	UF : 1, UT : 1,		CONFIG : 'N U T, 0, 0, 1',
	X =  25.000  mm,	Y =  64.000  mm,	Z =   15.000 mm,
	W =180.000 deg,	P =   0.000 deg,	R =    90.000 deg
};
P[3598]{
   GP1:
	UF : 1, UT : 1,		CONFIG : 'N U T, 0, 0, 1',
	X =  31.000  mm,	Y =  64.000  mm,	Z =   15.000 mm,
	W =180.000 deg,	P =   0.000 deg,	R =    90.000 deg
};
P[3599]{
   GP1:
	UF : 1, UT : 1,		CONFIG : 'N U T, 0, 0, 1',
	X =  31.000  mm,	Y =  64.000  mm,	Z =   0.600 mm,
	W =180.000 deg,	P =   0.000 deg,	R =    90.000 deg
};
P[3600]{
   GP1:
	UF : 1, UT : 1,		CONFIG : 'N U T, 0, 0, 1',
	X =  31.000  mm,	Y =  64.000  mm,	Z =   15.000 mm,
	W =180.000 deg,	P =   0.000 deg,	R =    90.000 deg
};
P[3601]{
   GP1:
	UF : 1, UT : 1,		CONFIG : 'N U T, 0, 0, 1',
	X =  34.000  mm,	Y =  64.000  mm,	Z =   15.000 mm,
	W =180.000 deg,	P =   0.000 deg,	R =    90.000 deg
};
P[3602]{
   GP1:
	UF : 1, UT : 1,		CONFIG : 'N U T, 0, 0, 1',
	X =  34.000  mm,	Y =  64.000  mm,	Z =   0.600 mm,
	W =180.000 deg,	P =   0.000 deg,	R =    90.000 deg
};
P[3603]{
   GP1:
	UF : 1, UT : 1,		CONFIG : 'N U T, 0, 0, 1',
	X =  34.000  mm,	Y =  64.000  mm,	Z =   15.000 mm,
	W =180.000 deg,	P =   0.000 deg,	R =    90.000 deg
};
P[3604]{
   GP1:
	UF : 1, UT : 1,		CONFIG : 'N U T, 0, 0, 1',
	X =  37.000  mm,	Y =  64.000  mm,	Z =   15.000 mm,
	W =180.000 deg,	P =   0.000 deg,	R =    90.000 deg
};
P[3605]{
   GP1:
	UF : 1, UT : 1,		CONFIG : 'N U T, 0, 0, 1',
	X =  37.000  mm,	Y =  64.000  mm,	Z =   0.600 mm,
	W =180.000 deg,	P =   0.000 deg,	R =    90.000 deg
};
P[3606]{
   GP1:
	UF : 1, UT : 1,		CONFIG : 'N U T, 0, 0, 1',
	X =  37.000  mm,	Y =  64.000  mm,	Z =   15.000 mm,
	W =180.000 deg,	P =   0.000 deg,	R =    90.000 deg
};
P[3607]{
   GP1:
	UF : 1, UT : 1,		CONFIG : 'N U T, 0, 0, 1',
	X =  40.000  mm,	Y =  64.000  mm,	Z =   15.000 mm,
	W =180.000 deg,	P =   0.000 deg,	R =    90.000 deg
};
P[3608]{
   GP1:
	UF : 1, UT : 1,		CONFIG : 'N U T, 0, 0, 1',
	X =  40.000  mm,	Y =  64.000  mm,	Z =   0.600 mm,
	W =180.000 deg,	P =   0.000 deg,	R =    90.000 deg
};
P[3609]{
   GP1:
	UF : 1, UT : 1,		CONFIG : 'N U T, 0, 0, 1',
	X =  40.000  mm,	Y =  64.000  mm,	Z =   15.000 mm,
	W =180.000 deg,	P =   0.000 deg,	R =    90.000 deg
};
P[3610]{
   GP1:
	UF : 1, UT : 1,		CONFIG : 'N U T, 0, 0, 1',
	X =  43.000  mm,	Y =  64.000  mm,	Z =   15.000 mm,
	W =180.000 deg,	P =   0.000 deg,	R =    90.000 deg
};
P[3611]{
   GP1:
	UF : 1, UT : 1,		CONFIG : 'N U T, 0, 0, 1',
	X =  43.000  mm,	Y =  64.000  mm,	Z =   0.600 mm,
	W =180.000 deg,	P =   0.000 deg,	R =    90.000 deg
};
P[3612]{
   GP1:
	UF : 1, UT : 1,		CONFIG : 'N U T, 0, 0, 1',
	X =  43.000  mm,	Y =  64.000  mm,	Z =   15.000 mm,
	W =180.000 deg,	P =   0.000 deg,	R =    90.000 deg
};
P[3613]{
   GP1:
	UF : 1, UT : 1,		CONFIG : 'N U T, 0, 0, 1',
	X =  46.000  mm,	Y =  64.000  mm,	Z =   15.000 mm,
	W =180.000 deg,	P =   0.000 deg,	R =    90.000 deg
};
P[3614]{
   GP1:
	UF : 1, UT : 1,		CONFIG : 'N U T, 0, 0, 1',
	X =  46.000  mm,	Y =  64.000  mm,	Z =   0.600 mm,
	W =180.000 deg,	P =   0.000 deg,	R =    90.000 deg
};
P[3615]{
   GP1:
	UF : 1, UT : 1,		CONFIG : 'N U T, 0, 0, 1',
	X =  46.000  mm,	Y =  64.000  mm,	Z =   15.000 mm,
	W =180.000 deg,	P =   0.000 deg,	R =    90.000 deg
};
P[3616]{
   GP1:
	UF : 1, UT : 1,		CONFIG : 'N U T, 0, 0, 1',
	X =  49.000  mm,	Y =  64.000  mm,	Z =   15.000 mm,
	W =180.000 deg,	P =   0.000 deg,	R =    90.000 deg
};
P[3617]{
   GP1:
	UF : 1, UT : 1,		CONFIG : 'N U T, 0, 0, 1',
	X =  49.000  mm,	Y =  64.000  mm,	Z =   0.600 mm,
	W =180.000 deg,	P =   0.000 deg,	R =    90.000 deg
};
P[3618]{
   GP1:
	UF : 1, UT : 1,		CONFIG : 'N U T, 0, 0, 1',
	X =  49.000  mm,	Y =  64.000  mm,	Z =   15.000 mm,
	W =180.000 deg,	P =   0.000 deg,	R =    90.000 deg
};
P[3619]{
   GP1:
	UF : 1, UT : 1,		CONFIG : 'N U T, 0, 0, 1',
	X =  52.000  mm,	Y =  64.000  mm,	Z =   15.000 mm,
	W =180.000 deg,	P =   0.000 deg,	R =    90.000 deg
};
P[3620]{
   GP1:
	UF : 1, UT : 1,		CONFIG : 'N U T, 0, 0, 1',
	X =  52.000  mm,	Y =  64.000  mm,	Z =   0.600 mm,
	W =180.000 deg,	P =   0.000 deg,	R =    90.000 deg
};
P[3621]{
   GP1:
	UF : 1, UT : 1,		CONFIG : 'N U T, 0, 0, 1',
	X =  52.000  mm,	Y =  64.000  mm,	Z =   15.000 mm,
	W =180.000 deg,	P =   0.000 deg,	R =    90.000 deg
};
P[3622]{
   GP1:
	UF : 1, UT : 1,		CONFIG : 'N U T, 0, 0, 1',
	X =  55.000  mm,	Y =  64.000  mm,	Z =   15.000 mm,
	W =180.000 deg,	P =   0.000 deg,	R =    90.000 deg
};
P[3623]{
   GP1:
	UF : 1, UT : 1,		CONFIG : 'N U T, 0, 0, 1',
	X =  55.000  mm,	Y =  64.000  mm,	Z =   0.600 mm,
	W =180.000 deg,	P =   0.000 deg,	R =    90.000 deg
};
P[3624]{
   GP1:
	UF : 1, UT : 1,		CONFIG : 'N U T, 0, 0, 1',
	X =  55.000  mm,	Y =  64.000  mm,	Z =   15.000 mm,
	W =180.000 deg,	P =   0.000 deg,	R =    90.000 deg
};
P[3628]{
   GP1:
	UF : 1, UT : 1,		CONFIG : 'N U T, 0, 0, 1',
	X =  61.000  mm,	Y =  64.000  mm,	Z =   15.000 mm,
	W =180.000 deg,	P =   0.000 deg,	R =    90.000 deg
};
P[3629]{
   GP1:
	UF : 1, UT : 1,		CONFIG : 'N U T, 0, 0, 1',
	X =  61.000  mm,	Y =  64.000  mm,	Z =   0.600 mm,
	W =180.000 deg,	P =   0.000 deg,	R =    90.000 deg
};
P[3630]{
   GP1:
	UF : 1, UT : 1,		CONFIG : 'N U T, 0, 0, 1',
	X =  61.000  mm,	Y =  64.000  mm,	Z =   15.000 mm,
	W =180.000 deg,	P =   0.000 deg,	R =    90.000 deg
};
P[3649]{
   GP1:
	UF : 1, UT : 1,		CONFIG : 'N U T, 0, 0, 1',
	X =  82.000  mm,	Y =  64.000  mm,	Z =   15.000 mm,
	W =180.000 deg,	P =   0.000 deg,	R =    90.000 deg
};
P[3650]{
   GP1:
	UF : 1, UT : 1,		CONFIG : 'N U T, 0, 0, 1',
	X =  82.000  mm,	Y =  64.000  mm,	Z =   0.600 mm,
	W =180.000 deg,	P =   0.000 deg,	R =    90.000 deg
};
P[3651]{
   GP1:
	UF : 1, UT : 1,		CONFIG : 'N U T, 0, 0, 1',
	X =  82.000  mm,	Y =  64.000  mm,	Z =   15.000 mm,
	W =180.000 deg,	P =   0.000 deg,	R =    90.000 deg
};
P[3652]{
   GP1:
	UF : 1, UT : 1,		CONFIG : 'N U T, 0, 0, 1',
	X =  85.000  mm,	Y =  64.000  mm,	Z =   15.000 mm,
	W =180.000 deg,	P =   0.000 deg,	R =    90.000 deg
};
P[3653]{
   GP1:
	UF : 1, UT : 1,		CONFIG : 'N U T, 0, 0, 1',
	X =  85.000  mm,	Y =  64.000  mm,	Z =   0.600 mm,
	W =180.000 deg,	P =   0.000 deg,	R =    90.000 deg
};
P[3654]{
   GP1:
	UF : 1, UT : 1,		CONFIG : 'N U T, 0, 0, 1',
	X =  85.000  mm,	Y =  64.000  mm,	Z =   15.000 mm,
	W =180.000 deg,	P =   0.000 deg,	R =    90.000 deg
};
P[3655]{
   GP1:
	UF : 1, UT : 1,		CONFIG : 'N U T, 0, 0, 1',
	X =  88.000  mm,	Y =  64.000  mm,	Z =   15.000 mm,
	W =180.000 deg,	P =   0.000 deg,	R =    90.000 deg
};
P[3656]{
   GP1:
	UF : 1, UT : 1,		CONFIG : 'N U T, 0, 0, 1',
	X =  88.000  mm,	Y =  64.000  mm,	Z =   0.600 mm,
	W =180.000 deg,	P =   0.000 deg,	R =    90.000 deg
};
P[3657]{
   GP1:
	UF : 1, UT : 1,		CONFIG : 'N U T, 0, 0, 1',
	X =  88.000  mm,	Y =  64.000  mm,	Z =   15.000 mm,
	W =180.000 deg,	P =   0.000 deg,	R =    90.000 deg
};
P[3658]{
   GP1:
	UF : 1, UT : 1,		CONFIG : 'N U T, 0, 0, 1',
	X =  91.000  mm,	Y =  64.000  mm,	Z =   15.000 mm,
	W =180.000 deg,	P =   0.000 deg,	R =    90.000 deg
};
P[3659]{
   GP1:
	UF : 1, UT : 1,		CONFIG : 'N U T, 0, 0, 1',
	X =  91.000  mm,	Y =  64.000  mm,	Z =   0.600 mm,
	W =180.000 deg,	P =   0.000 deg,	R =    90.000 deg
};
P[3660]{
   GP1:
	UF : 1, UT : 1,		CONFIG : 'N U T, 0, 0, 1',
	X =  91.000  mm,	Y =  64.000  mm,	Z =   15.000 mm,
	W =180.000 deg,	P =   0.000 deg,	R =    90.000 deg
};
P[3661]{
   GP1:
	UF : 1, UT : 1,		CONFIG : 'N U T, 0, 0, 1',
	X =  94.000  mm,	Y =  64.000  mm,	Z =   15.000 mm,
	W =180.000 deg,	P =   0.000 deg,	R =    90.000 deg
};
P[3662]{
   GP1:
	UF : 1, UT : 1,		CONFIG : 'N U T, 0, 0, 1',
	X =  94.000  mm,	Y =  64.000  mm,	Z =   0.600 mm,
	W =180.000 deg,	P =   0.000 deg,	R =    90.000 deg
};
P[3663]{
   GP1:
	UF : 1, UT : 1,		CONFIG : 'N U T, 0, 0, 1',
	X =  94.000  mm,	Y =  64.000  mm,	Z =   15.000 mm,
	W =180.000 deg,	P =   0.000 deg,	R =    90.000 deg
};
P[3664]{
   GP1:
	UF : 1, UT : 1,		CONFIG : 'N U T, 0, 0, 1',
	X =  97.000  mm,	Y =  64.000  mm,	Z =   15.000 mm,
	W =180.000 deg,	P =   0.000 deg,	R =    90.000 deg
};
P[3665]{
   GP1:
	UF : 1, UT : 1,		CONFIG : 'N U T, 0, 0, 1',
	X =  97.000  mm,	Y =  64.000  mm,	Z =   0.600 mm,
	W =180.000 deg,	P =   0.000 deg,	R =    90.000 deg
};
P[3666]{
   GP1:
	UF : 1, UT : 1,		CONFIG : 'N U T, 0, 0, 1',
	X =  97.000  mm,	Y =  64.000  mm,	Z =   15.000 mm,
	W =180.000 deg,	P =   0.000 deg,	R =    90.000 deg
};
P[3667]{
   GP1:
	UF : 1, UT : 1,		CONFIG : 'N U T, 0, 0, 1',
	X =  100.000  mm,	Y =  64.000  mm,	Z =   15.000 mm,
	W =180.000 deg,	P =   0.000 deg,	R =    90.000 deg
};
P[3668]{
   GP1:
	UF : 1, UT : 1,		CONFIG : 'N U T, 0, 0, 1',
	X =  100.000  mm,	Y =  64.000  mm,	Z =   0.600 mm,
	W =180.000 deg,	P =   0.000 deg,	R =    90.000 deg
};
P[3669]{
   GP1:
	UF : 1, UT : 1,		CONFIG : 'N U T, 0, 0, 1',
	X =  100.000  mm,	Y =  64.000  mm,	Z =   15.000 mm,
	W =180.000 deg,	P =   0.000 deg,	R =    90.000 deg
};
P[3670]{
   GP1:
	UF : 1, UT : 1,		CONFIG : 'N U T, 0, 0, 1',
	X =  103.000  mm,	Y =  64.000  mm,	Z =   15.000 mm,
	W =180.000 deg,	P =   0.000 deg,	R =    90.000 deg
};
P[3671]{
   GP1:
	UF : 1, UT : 1,		CONFIG : 'N U T, 0, 0, 1',
	X =  103.000  mm,	Y =  64.000  mm,	Z =   0.600 mm,
	W =180.000 deg,	P =   0.000 deg,	R =    90.000 deg
};
P[3672]{
   GP1:
	UF : 1, UT : 1,		CONFIG : 'N U T, 0, 0, 1',
	X =  103.000  mm,	Y =  64.000  mm,	Z =   15.000 mm,
	W =180.000 deg,	P =   0.000 deg,	R =    90.000 deg
};
P[3673]{
   GP1:
	UF : 1, UT : 1,		CONFIG : 'N U T, 0, 0, 1',
	X =  106.000  mm,	Y =  64.000  mm,	Z =   15.000 mm,
	W =180.000 deg,	P =   0.000 deg,	R =    90.000 deg
};
P[3674]{
   GP1:
	UF : 1, UT : 1,		CONFIG : 'N U T, 0, 0, 1',
	X =  106.000  mm,	Y =  64.000  mm,	Z =   0.600 mm,
	W =180.000 deg,	P =   0.000 deg,	R =    90.000 deg
};
P[3675]{
   GP1:
	UF : 1, UT : 1,		CONFIG : 'N U T, 0, 0, 1',
	X =  106.000  mm,	Y =  64.000  mm,	Z =   15.000 mm,
	W =180.000 deg,	P =   0.000 deg,	R =    90.000 deg
};
P[3676]{
   GP1:
	UF : 1, UT : 1,		CONFIG : 'N U T, 0, 0, 1',
	X =  109.000  mm,	Y =  64.000  mm,	Z =   15.000 mm,
	W =180.000 deg,	P =   0.000 deg,	R =    90.000 deg
};
P[3677]{
   GP1:
	UF : 1, UT : 1,		CONFIG : 'N U T, 0, 0, 1',
	X =  109.000  mm,	Y =  64.000  mm,	Z =   0.600 mm,
	W =180.000 deg,	P =   0.000 deg,	R =    90.000 deg
};
P[3678]{
   GP1:
	UF : 1, UT : 1,		CONFIG : 'N U T, 0, 0, 1',
	X =  109.000  mm,	Y =  64.000  mm,	Z =   15.000 mm,
	W =180.000 deg,	P =   0.000 deg,	R =    90.000 deg
};
P[3679]{
   GP1:
	UF : 1, UT : 1,		CONFIG : 'N U T, 0, 0, 1',
	X =  112.000  mm,	Y =  64.000  mm,	Z =   15.000 mm,
	W =180.000 deg,	P =   0.000 deg,	R =    90.000 deg
};
P[3680]{
   GP1:
	UF : 1, UT : 1,		CONFIG : 'N U T, 0, 0, 1',
	X =  112.000  mm,	Y =  64.000  mm,	Z =   0.600 mm,
	W =180.000 deg,	P =   0.000 deg,	R =    90.000 deg
};
P[3681]{
   GP1:
	UF : 1, UT : 1,		CONFIG : 'N U T, 0, 0, 1',
	X =  112.000  mm,	Y =  64.000  mm,	Z =   15.000 mm,
	W =180.000 deg,	P =   0.000 deg,	R =    90.000 deg
};
P[3682]{
   GP1:
	UF : 1, UT : 1,		CONFIG : 'N U T, 0, 0, 1',
	X =  115.000  mm,	Y =  64.000  mm,	Z =   15.000 mm,
	W =180.000 deg,	P =   0.000 deg,	R =    90.000 deg
};
P[3683]{
   GP1:
	UF : 1, UT : 1,		CONFIG : 'N U T, 0, 0, 1',
	X =  115.000  mm,	Y =  64.000  mm,	Z =   0.600 mm,
	W =180.000 deg,	P =   0.000 deg,	R =    90.000 deg
};
P[3684]{
   GP1:
	UF : 1, UT : 1,		CONFIG : 'N U T, 0, 0, 1',
	X =  115.000  mm,	Y =  64.000  mm,	Z =   15.000 mm,
	W =180.000 deg,	P =   0.000 deg,	R =    90.000 deg
};
P[3691]{
   GP1:
	UF : 1, UT : 1,		CONFIG : 'N U T, 0, 0, 1',
	X =  130.000  mm,	Y =  64.000  mm,	Z =   15.000 mm,
	W =180.000 deg,	P =   0.000 deg,	R =    90.000 deg
};
P[3692]{
   GP1:
	UF : 1, UT : 1,		CONFIG : 'N U T, 0, 0, 1',
	X =  130.000  mm,	Y =  64.000  mm,	Z =   0.600 mm,
	W =180.000 deg,	P =   0.000 deg,	R =    90.000 deg
};
P[3693]{
   GP1:
	UF : 1, UT : 1,		CONFIG : 'N U T, 0, 0, 1',
	X =  130.000  mm,	Y =  64.000  mm,	Z =   15.000 mm,
	W =180.000 deg,	P =   0.000 deg,	R =    90.000 deg
};
P[3703]{
   GP1:
	UF : 1, UT : 1,		CONFIG : 'N U T, 0, 0, 1',
	X =  142.000  mm,	Y =  64.000  mm,	Z =   15.000 mm,
	W =180.000 deg,	P =   0.000 deg,	R =    90.000 deg
};
P[3704]{
   GP1:
	UF : 1, UT : 1,		CONFIG : 'N U T, 0, 0, 1',
	X =  142.000  mm,	Y =  64.000  mm,	Z =   0.600 mm,
	W =180.000 deg,	P =   0.000 deg,	R =    90.000 deg
};
P[3705]{
   GP1:
	UF : 1, UT : 1,		CONFIG : 'N U T, 0, 0, 1',
	X =  142.000  mm,	Y =  64.000  mm,	Z =   15.000 mm,
	W =180.000 deg,	P =   0.000 deg,	R =    90.000 deg
};
P[3706]{
   GP1:
	UF : 1, UT : 1,		CONFIG : 'N U T, 0, 0, 1',
	X =  145.000  mm,	Y =  64.000  mm,	Z =   15.000 mm,
	W =180.000 deg,	P =   0.000 deg,	R =    90.000 deg
};
P[3707]{
   GP1:
	UF : 1, UT : 1,		CONFIG : 'N U T, 0, 0, 1',
	X =  145.000  mm,	Y =  64.000  mm,	Z =   0.600 mm,
	W =180.000 deg,	P =   0.000 deg,	R =    90.000 deg
};
P[3708]{
   GP1:
	UF : 1, UT : 1,		CONFIG : 'N U T, 0, 0, 1',
	X =  145.000  mm,	Y =  64.000  mm,	Z =   15.000 mm,
	W =180.000 deg,	P =   0.000 deg,	R =    90.000 deg
};
P[3709]{
   GP1:
	UF : 1, UT : 1,		CONFIG : 'N U T, 0, 0, 1',
	X =  172.000  mm,	Y =  64.000  mm,	Z =   15.000 mm,
	W =180.000 deg,	P =   0.000 deg,	R =    90.000 deg
};
P[3710]{
   GP1:
	UF : 1, UT : 1,		CONFIG : 'N U T, 0, 0, 1',
	X =  172.000  mm,	Y =  64.000  mm,	Z =   0.600 mm,
	W =180.000 deg,	P =   0.000 deg,	R =    90.000 deg
};
P[3711]{
   GP1:
	UF : 1, UT : 1,		CONFIG : 'N U T, 0, 0, 1',
	X =  172.000  mm,	Y =  64.000  mm,	Z =   15.000 mm,
	W =180.000 deg,	P =   0.000 deg,	R =    90.000 deg
};
P[3712]{
   GP1:
	UF : 1, UT : 1,		CONFIG : 'N U T, 0, 0, 1',
	X =  175.000  mm,	Y =  64.000  mm,	Z =   15.000 mm,
	W =180.000 deg,	P =   0.000 deg,	R =    90.000 deg
};
P[3713]{
   GP1:
	UF : 1, UT : 1,		CONFIG : 'N U T, 0, 0, 1',
	X =  175.000  mm,	Y =  64.000  mm,	Z =   0.600 mm,
	W =180.000 deg,	P =   0.000 deg,	R =    90.000 deg
};
P[3714]{
   GP1:
	UF : 1, UT : 1,		CONFIG : 'N U T, 0, 0, 1',
	X =  175.000  mm,	Y =  64.000  mm,	Z =   15.000 mm,
	W =180.000 deg,	P =   0.000 deg,	R =    90.000 deg
};
P[3715]{
   GP1:
	UF : 1, UT : 1,		CONFIG : 'N U T, 0, 0, 1',
	X =  178.000  mm,	Y =  64.000  mm,	Z =   15.000 mm,
	W =180.000 deg,	P =   0.000 deg,	R =    90.000 deg
};
P[3716]{
   GP1:
	UF : 1, UT : 1,		CONFIG : 'N U T, 0, 0, 1',
	X =  178.000  mm,	Y =  64.000  mm,	Z =   0.600 mm,
	W =180.000 deg,	P =   0.000 deg,	R =    90.000 deg
};
P[3717]{
   GP1:
	UF : 1, UT : 1,		CONFIG : 'N U T, 0, 0, 1',
	X =  178.000  mm,	Y =  64.000  mm,	Z =   15.000 mm,
	W =180.000 deg,	P =   0.000 deg,	R =    90.000 deg
};
P[3718]{
   GP1:
	UF : 1, UT : 1,		CONFIG : 'N U T, 0, 0, 1',
	X =  1.000  mm,	Y =  67.000  mm,	Z =   15.000 mm,
	W =180.000 deg,	P =   0.000 deg,	R =    90.000 deg
};
P[3719]{
   GP1:
	UF : 1, UT : 1,		CONFIG : 'N U T, 0, 0, 1',
	X =  1.000  mm,	Y =  67.000  mm,	Z =   0.600 mm,
	W =180.000 deg,	P =   0.000 deg,	R =    90.000 deg
};
P[3720]{
   GP1:
	UF : 1, UT : 1,		CONFIG : 'N U T, 0, 0, 1',
	X =  1.000  mm,	Y =  67.000  mm,	Z =   15.000 mm,
	W =180.000 deg,	P =   0.000 deg,	R =    90.000 deg
};
P[3721]{
   GP1:
	UF : 1, UT : 1,		CONFIG : 'N U T, 0, 0, 1',
	X =  4.000  mm,	Y =  67.000  mm,	Z =   15.000 mm,
	W =180.000 deg,	P =   0.000 deg,	R =    90.000 deg
};
P[3722]{
   GP1:
	UF : 1, UT : 1,		CONFIG : 'N U T, 0, 0, 1',
	X =  4.000  mm,	Y =  67.000  mm,	Z =   0.600 mm,
	W =180.000 deg,	P =   0.000 deg,	R =    90.000 deg
};
P[3723]{
   GP1:
	UF : 1, UT : 1,		CONFIG : 'N U T, 0, 0, 1',
	X =  4.000  mm,	Y =  67.000  mm,	Z =   15.000 mm,
	W =180.000 deg,	P =   0.000 deg,	R =    90.000 deg
};
P[3724]{
   GP1:
	UF : 1, UT : 1,		CONFIG : 'N U T, 0, 0, 1',
	X =  7.000  mm,	Y =  67.000  mm,	Z =   15.000 mm,
	W =180.000 deg,	P =   0.000 deg,	R =    90.000 deg
};
P[3725]{
   GP1:
	UF : 1, UT : 1,		CONFIG : 'N U T, 0, 0, 1',
	X =  7.000  mm,	Y =  67.000  mm,	Z =   0.600 mm,
	W =180.000 deg,	P =   0.000 deg,	R =    90.000 deg
};
P[3726]{
   GP1:
	UF : 1, UT : 1,		CONFIG : 'N U T, 0, 0, 1',
	X =  7.000  mm,	Y =  67.000  mm,	Z =   15.000 mm,
	W =180.000 deg,	P =   0.000 deg,	R =    90.000 deg
};
P[3727]{
   GP1:
	UF : 1, UT : 1,		CONFIG : 'N U T, 0, 0, 1',
	X =  10.000  mm,	Y =  67.000  mm,	Z =   15.000 mm,
	W =180.000 deg,	P =   0.000 deg,	R =    90.000 deg
};
P[3728]{
   GP1:
	UF : 1, UT : 1,		CONFIG : 'N U T, 0, 0, 1',
	X =  10.000  mm,	Y =  67.000  mm,	Z =   0.600 mm,
	W =180.000 deg,	P =   0.000 deg,	R =    90.000 deg
};
P[3729]{
   GP1:
	UF : 1, UT : 1,		CONFIG : 'N U T, 0, 0, 1',
	X =  10.000  mm,	Y =  67.000  mm,	Z =   15.000 mm,
	W =180.000 deg,	P =   0.000 deg,	R =    90.000 deg
};
P[3730]{
   GP1:
	UF : 1, UT : 1,		CONFIG : 'N U T, 0, 0, 1',
	X =  13.000  mm,	Y =  67.000  mm,	Z =   15.000 mm,
	W =180.000 deg,	P =   0.000 deg,	R =    90.000 deg
};
P[3731]{
   GP1:
	UF : 1, UT : 1,		CONFIG : 'N U T, 0, 0, 1',
	X =  13.000  mm,	Y =  67.000  mm,	Z =   0.600 mm,
	W =180.000 deg,	P =   0.000 deg,	R =    90.000 deg
};
P[3732]{
   GP1:
	UF : 1, UT : 1,		CONFIG : 'N U T, 0, 0, 1',
	X =  13.000  mm,	Y =  67.000  mm,	Z =   15.000 mm,
	W =180.000 deg,	P =   0.000 deg,	R =    90.000 deg
};
P[3733]{
   GP1:
	UF : 1, UT : 1,		CONFIG : 'N U T, 0, 0, 1',
	X =  16.000  mm,	Y =  67.000  mm,	Z =   15.000 mm,
	W =180.000 deg,	P =   0.000 deg,	R =    90.000 deg
};
P[3734]{
   GP1:
	UF : 1, UT : 1,		CONFIG : 'N U T, 0, 0, 1',
	X =  16.000  mm,	Y =  67.000  mm,	Z =   0.600 mm,
	W =180.000 deg,	P =   0.000 deg,	R =    90.000 deg
};
P[3735]{
   GP1:
	UF : 1, UT : 1,		CONFIG : 'N U T, 0, 0, 1',
	X =  16.000  mm,	Y =  67.000  mm,	Z =   15.000 mm,
	W =180.000 deg,	P =   0.000 deg,	R =    90.000 deg
};
P[3736]{
   GP1:
	UF : 1, UT : 1,		CONFIG : 'N U T, 0, 0, 1',
	X =  19.000  mm,	Y =  67.000  mm,	Z =   15.000 mm,
	W =180.000 deg,	P =   0.000 deg,	R =    90.000 deg
};
P[3737]{
   GP1:
	UF : 1, UT : 1,		CONFIG : 'N U T, 0, 0, 1',
	X =  19.000  mm,	Y =  67.000  mm,	Z =   0.600 mm,
	W =180.000 deg,	P =   0.000 deg,	R =    90.000 deg
};
P[3738]{
   GP1:
	UF : 1, UT : 1,		CONFIG : 'N U T, 0, 0, 1',
	X =  19.000  mm,	Y =  67.000  mm,	Z =   15.000 mm,
	W =180.000 deg,	P =   0.000 deg,	R =    90.000 deg
};
P[3739]{
   GP1:
	UF : 1, UT : 1,		CONFIG : 'N U T, 0, 0, 1',
	X =  22.000  mm,	Y =  67.000  mm,	Z =   15.000 mm,
	W =180.000 deg,	P =   0.000 deg,	R =    90.000 deg
};
P[3740]{
   GP1:
	UF : 1, UT : 1,		CONFIG : 'N U T, 0, 0, 1',
	X =  22.000  mm,	Y =  67.000  mm,	Z =   0.600 mm,
	W =180.000 deg,	P =   0.000 deg,	R =    90.000 deg
};
P[3741]{
   GP1:
	UF : 1, UT : 1,		CONFIG : 'N U T, 0, 0, 1',
	X =  22.000  mm,	Y =  67.000  mm,	Z =   15.000 mm,
	W =180.000 deg,	P =   0.000 deg,	R =    90.000 deg
};
P[3742]{
   GP1:
	UF : 1, UT : 1,		CONFIG : 'N U T, 0, 0, 1',
	X =  25.000  mm,	Y =  67.000  mm,	Z =   15.000 mm,
	W =180.000 deg,	P =   0.000 deg,	R =    90.000 deg
};
P[3743]{
   GP1:
	UF : 1, UT : 1,		CONFIG : 'N U T, 0, 0, 1',
	X =  25.000  mm,	Y =  67.000  mm,	Z =   0.600 mm,
	W =180.000 deg,	P =   0.000 deg,	R =    90.000 deg
};
P[3744]{
   GP1:
	UF : 1, UT : 1,		CONFIG : 'N U T, 0, 0, 1',
	X =  25.000  mm,	Y =  67.000  mm,	Z =   15.000 mm,
	W =180.000 deg,	P =   0.000 deg,	R =    90.000 deg
};
P[3745]{
   GP1:
	UF : 1, UT : 1,		CONFIG : 'N U T, 0, 0, 1',
	X =  34.000  mm,	Y =  67.000  mm,	Z =   15.000 mm,
	W =180.000 deg,	P =   0.000 deg,	R =    90.000 deg
};
P[3746]{
   GP1:
	UF : 1, UT : 1,		CONFIG : 'N U T, 0, 0, 1',
	X =  34.000  mm,	Y =  67.000  mm,	Z =   0.600 mm,
	W =180.000 deg,	P =   0.000 deg,	R =    90.000 deg
};
P[3747]{
   GP1:
	UF : 1, UT : 1,		CONFIG : 'N U T, 0, 0, 1',
	X =  34.000  mm,	Y =  67.000  mm,	Z =   15.000 mm,
	W =180.000 deg,	P =   0.000 deg,	R =    90.000 deg
};
P[3748]{
   GP1:
	UF : 1, UT : 1,		CONFIG : 'N U T, 0, 0, 1',
	X =  37.000  mm,	Y =  67.000  mm,	Z =   15.000 mm,
	W =180.000 deg,	P =   0.000 deg,	R =    90.000 deg
};
P[3749]{
   GP1:
	UF : 1, UT : 1,		CONFIG : 'N U T, 0, 0, 1',
	X =  37.000  mm,	Y =  67.000  mm,	Z =   0.600 mm,
	W =180.000 deg,	P =   0.000 deg,	R =    90.000 deg
};
P[3750]{
   GP1:
	UF : 1, UT : 1,		CONFIG : 'N U T, 0, 0, 1',
	X =  37.000  mm,	Y =  67.000  mm,	Z =   15.000 mm,
	W =180.000 deg,	P =   0.000 deg,	R =    90.000 deg
};
P[3751]{
   GP1:
	UF : 1, UT : 1,		CONFIG : 'N U T, 0, 0, 1',
	X =  40.000  mm,	Y =  67.000  mm,	Z =   15.000 mm,
	W =180.000 deg,	P =   0.000 deg,	R =    90.000 deg
};
P[3752]{
   GP1:
	UF : 1, UT : 1,		CONFIG : 'N U T, 0, 0, 1',
	X =  40.000  mm,	Y =  67.000  mm,	Z =   0.600 mm,
	W =180.000 deg,	P =   0.000 deg,	R =    90.000 deg
};
P[3753]{
   GP1:
	UF : 1, UT : 1,		CONFIG : 'N U T, 0, 0, 1',
	X =  40.000  mm,	Y =  67.000  mm,	Z =   15.000 mm,
	W =180.000 deg,	P =   0.000 deg,	R =    90.000 deg
};
P[3754]{
   GP1:
	UF : 1, UT : 1,		CONFIG : 'N U T, 0, 0, 1',
	X =  43.000  mm,	Y =  67.000  mm,	Z =   15.000 mm,
	W =180.000 deg,	P =   0.000 deg,	R =    90.000 deg
};
P[3755]{
   GP1:
	UF : 1, UT : 1,		CONFIG : 'N U T, 0, 0, 1',
	X =  43.000  mm,	Y =  67.000  mm,	Z =   0.600 mm,
	W =180.000 deg,	P =   0.000 deg,	R =    90.000 deg
};
P[3756]{
   GP1:
	UF : 1, UT : 1,		CONFIG : 'N U T, 0, 0, 1',
	X =  43.000  mm,	Y =  67.000  mm,	Z =   15.000 mm,
	W =180.000 deg,	P =   0.000 deg,	R =    90.000 deg
};
P[3757]{
   GP1:
	UF : 1, UT : 1,		CONFIG : 'N U T, 0, 0, 1',
	X =  46.000  mm,	Y =  67.000  mm,	Z =   15.000 mm,
	W =180.000 deg,	P =   0.000 deg,	R =    90.000 deg
};
P[3758]{
   GP1:
	UF : 1, UT : 1,		CONFIG : 'N U T, 0, 0, 1',
	X =  46.000  mm,	Y =  67.000  mm,	Z =   0.600 mm,
	W =180.000 deg,	P =   0.000 deg,	R =    90.000 deg
};
P[3759]{
   GP1:
	UF : 1, UT : 1,		CONFIG : 'N U T, 0, 0, 1',
	X =  46.000  mm,	Y =  67.000  mm,	Z =   15.000 mm,
	W =180.000 deg,	P =   0.000 deg,	R =    90.000 deg
};
P[3760]{
   GP1:
	UF : 1, UT : 1,		CONFIG : 'N U T, 0, 0, 1',
	X =  49.000  mm,	Y =  67.000  mm,	Z =   15.000 mm,
	W =180.000 deg,	P =   0.000 deg,	R =    90.000 deg
};
P[3761]{
   GP1:
	UF : 1, UT : 1,		CONFIG : 'N U T, 0, 0, 1',
	X =  49.000  mm,	Y =  67.000  mm,	Z =   0.600 mm,
	W =180.000 deg,	P =   0.000 deg,	R =    90.000 deg
};
P[3762]{
   GP1:
	UF : 1, UT : 1,		CONFIG : 'N U T, 0, 0, 1',
	X =  49.000  mm,	Y =  67.000  mm,	Z =   15.000 mm,
	W =180.000 deg,	P =   0.000 deg,	R =    90.000 deg
};
P[3763]{
   GP1:
	UF : 1, UT : 1,		CONFIG : 'N U T, 0, 0, 1',
	X =  52.000  mm,	Y =  67.000  mm,	Z =   15.000 mm,
	W =180.000 deg,	P =   0.000 deg,	R =    90.000 deg
};
P[3764]{
   GP1:
	UF : 1, UT : 1,		CONFIG : 'N U T, 0, 0, 1',
	X =  52.000  mm,	Y =  67.000  mm,	Z =   0.600 mm,
	W =180.000 deg,	P =   0.000 deg,	R =    90.000 deg
};
P[3765]{
   GP1:
	UF : 1, UT : 1,		CONFIG : 'N U T, 0, 0, 1',
	X =  52.000  mm,	Y =  67.000  mm,	Z =   15.000 mm,
	W =180.000 deg,	P =   0.000 deg,	R =    90.000 deg
};
P[3766]{
   GP1:
	UF : 1, UT : 1,		CONFIG : 'N U T, 0, 0, 1',
	X =  55.000  mm,	Y =  67.000  mm,	Z =   15.000 mm,
	W =180.000 deg,	P =   0.000 deg,	R =    90.000 deg
};
P[3767]{
   GP1:
	UF : 1, UT : 1,		CONFIG : 'N U T, 0, 0, 1',
	X =  55.000  mm,	Y =  67.000  mm,	Z =   0.600 mm,
	W =180.000 deg,	P =   0.000 deg,	R =    90.000 deg
};
P[3768]{
   GP1:
	UF : 1, UT : 1,		CONFIG : 'N U T, 0, 0, 1',
	X =  55.000  mm,	Y =  67.000  mm,	Z =   15.000 mm,
	W =180.000 deg,	P =   0.000 deg,	R =    90.000 deg
};
P[3769]{
   GP1:
	UF : 1, UT : 1,		CONFIG : 'N U T, 0, 0, 1',
	X =  58.000  mm,	Y =  67.000  mm,	Z =   15.000 mm,
	W =180.000 deg,	P =   0.000 deg,	R =    90.000 deg
};
P[3770]{
   GP1:
	UF : 1, UT : 1,		CONFIG : 'N U T, 0, 0, 1',
	X =  58.000  mm,	Y =  67.000  mm,	Z =   0.600 mm,
	W =180.000 deg,	P =   0.000 deg,	R =    90.000 deg
};
P[3771]{
   GP1:
	UF : 1, UT : 1,		CONFIG : 'N U T, 0, 0, 1',
	X =  58.000  mm,	Y =  67.000  mm,	Z =   15.000 mm,
	W =180.000 deg,	P =   0.000 deg,	R =    90.000 deg
};
P[3772]{
   GP1:
	UF : 1, UT : 1,		CONFIG : 'N U T, 0, 0, 1',
	X =  61.000  mm,	Y =  67.000  mm,	Z =   15.000 mm,
	W =180.000 deg,	P =   0.000 deg,	R =    90.000 deg
};
P[3773]{
   GP1:
	UF : 1, UT : 1,		CONFIG : 'N U T, 0, 0, 1',
	X =  61.000  mm,	Y =  67.000  mm,	Z =   0.600 mm,
	W =180.000 deg,	P =   0.000 deg,	R =    90.000 deg
};
P[3774]{
   GP1:
	UF : 1, UT : 1,		CONFIG : 'N U T, 0, 0, 1',
	X =  61.000  mm,	Y =  67.000  mm,	Z =   15.000 mm,
	W =180.000 deg,	P =   0.000 deg,	R =    90.000 deg
};
P[3790]{
   GP1:
	UF : 1, UT : 1,		CONFIG : 'N U T, 0, 0, 1',
	X =  79.000  mm,	Y =  67.000  mm,	Z =   15.000 mm,
	W =180.000 deg,	P =   0.000 deg,	R =    90.000 deg
};
P[3791]{
   GP1:
	UF : 1, UT : 1,		CONFIG : 'N U T, 0, 0, 1',
	X =  79.000  mm,	Y =  67.000  mm,	Z =   0.600 mm,
	W =180.000 deg,	P =   0.000 deg,	R =    90.000 deg
};
P[3792]{
   GP1:
	UF : 1, UT : 1,		CONFIG : 'N U T, 0, 0, 1',
	X =  79.000  mm,	Y =  67.000  mm,	Z =   15.000 mm,
	W =180.000 deg,	P =   0.000 deg,	R =    90.000 deg
};
P[3793]{
   GP1:
	UF : 1, UT : 1,		CONFIG : 'N U T, 0, 0, 1',
	X =  82.000  mm,	Y =  67.000  mm,	Z =   15.000 mm,
	W =180.000 deg,	P =   0.000 deg,	R =    90.000 deg
};
P[3794]{
   GP1:
	UF : 1, UT : 1,		CONFIG : 'N U T, 0, 0, 1',
	X =  82.000  mm,	Y =  67.000  mm,	Z =   0.600 mm,
	W =180.000 deg,	P =   0.000 deg,	R =    90.000 deg
};
P[3795]{
   GP1:
	UF : 1, UT : 1,		CONFIG : 'N U T, 0, 0, 1',
	X =  82.000  mm,	Y =  67.000  mm,	Z =   15.000 mm,
	W =180.000 deg,	P =   0.000 deg,	R =    90.000 deg
};
P[3796]{
   GP1:
	UF : 1, UT : 1,		CONFIG : 'N U T, 0, 0, 1',
	X =  85.000  mm,	Y =  67.000  mm,	Z =   15.000 mm,
	W =180.000 deg,	P =   0.000 deg,	R =    90.000 deg
};
P[3797]{
   GP1:
	UF : 1, UT : 1,		CONFIG : 'N U T, 0, 0, 1',
	X =  85.000  mm,	Y =  67.000  mm,	Z =   0.600 mm,
	W =180.000 deg,	P =   0.000 deg,	R =    90.000 deg
};
P[3798]{
   GP1:
	UF : 1, UT : 1,		CONFIG : 'N U T, 0, 0, 1',
	X =  85.000  mm,	Y =  67.000  mm,	Z =   15.000 mm,
	W =180.000 deg,	P =   0.000 deg,	R =    90.000 deg
};
P[3799]{
   GP1:
	UF : 1, UT : 1,		CONFIG : 'N U T, 0, 0, 1',
	X =  88.000  mm,	Y =  67.000  mm,	Z =   15.000 mm,
	W =180.000 deg,	P =   0.000 deg,	R =    90.000 deg
};
P[3800]{
   GP1:
	UF : 1, UT : 1,		CONFIG : 'N U T, 0, 0, 1',
	X =  88.000  mm,	Y =  67.000  mm,	Z =   0.600 mm,
	W =180.000 deg,	P =   0.000 deg,	R =    90.000 deg
};
P[3801]{
   GP1:
	UF : 1, UT : 1,		CONFIG : 'N U T, 0, 0, 1',
	X =  88.000  mm,	Y =  67.000  mm,	Z =   15.000 mm,
	W =180.000 deg,	P =   0.000 deg,	R =    90.000 deg
};
P[3802]{
   GP1:
	UF : 1, UT : 1,		CONFIG : 'N U T, 0, 0, 1',
	X =  91.000  mm,	Y =  67.000  mm,	Z =   15.000 mm,
	W =180.000 deg,	P =   0.000 deg,	R =    90.000 deg
};
P[3803]{
   GP1:
	UF : 1, UT : 1,		CONFIG : 'N U T, 0, 0, 1',
	X =  91.000  mm,	Y =  67.000  mm,	Z =   0.600 mm,
	W =180.000 deg,	P =   0.000 deg,	R =    90.000 deg
};
P[3804]{
   GP1:
	UF : 1, UT : 1,		CONFIG : 'N U T, 0, 0, 1',
	X =  91.000  mm,	Y =  67.000  mm,	Z =   15.000 mm,
	W =180.000 deg,	P =   0.000 deg,	R =    90.000 deg
};
P[3805]{
   GP1:
	UF : 1, UT : 1,		CONFIG : 'N U T, 0, 0, 1',
	X =  94.000  mm,	Y =  67.000  mm,	Z =   15.000 mm,
	W =180.000 deg,	P =   0.000 deg,	R =    90.000 deg
};
P[3806]{
   GP1:
	UF : 1, UT : 1,		CONFIG : 'N U T, 0, 0, 1',
	X =  94.000  mm,	Y =  67.000  mm,	Z =   0.600 mm,
	W =180.000 deg,	P =   0.000 deg,	R =    90.000 deg
};
P[3807]{
   GP1:
	UF : 1, UT : 1,		CONFIG : 'N U T, 0, 0, 1',
	X =  94.000  mm,	Y =  67.000  mm,	Z =   15.000 mm,
	W =180.000 deg,	P =   0.000 deg,	R =    90.000 deg
};
P[3808]{
   GP1:
	UF : 1, UT : 1,		CONFIG : 'N U T, 0, 0, 1',
	X =  97.000  mm,	Y =  67.000  mm,	Z =   15.000 mm,
	W =180.000 deg,	P =   0.000 deg,	R =    90.000 deg
};
P[3809]{
   GP1:
	UF : 1, UT : 1,		CONFIG : 'N U T, 0, 0, 1',
	X =  97.000  mm,	Y =  67.000  mm,	Z =   0.600 mm,
	W =180.000 deg,	P =   0.000 deg,	R =    90.000 deg
};
P[3810]{
   GP1:
	UF : 1, UT : 1,		CONFIG : 'N U T, 0, 0, 1',
	X =  97.000  mm,	Y =  67.000  mm,	Z =   15.000 mm,
	W =180.000 deg,	P =   0.000 deg,	R =    90.000 deg
};
P[3811]{
   GP1:
	UF : 1, UT : 1,		CONFIG : 'N U T, 0, 0, 1',
	X =  100.000  mm,	Y =  67.000  mm,	Z =   15.000 mm,
	W =180.000 deg,	P =   0.000 deg,	R =    90.000 deg
};
P[3812]{
   GP1:
	UF : 1, UT : 1,		CONFIG : 'N U T, 0, 0, 1',
	X =  100.000  mm,	Y =  67.000  mm,	Z =   0.600 mm,
	W =180.000 deg,	P =   0.000 deg,	R =    90.000 deg
};
P[3813]{
   GP1:
	UF : 1, UT : 1,		CONFIG : 'N U T, 0, 0, 1',
	X =  100.000  mm,	Y =  67.000  mm,	Z =   15.000 mm,
	W =180.000 deg,	P =   0.000 deg,	R =    90.000 deg
};
P[3814]{
   GP1:
	UF : 1, UT : 1,		CONFIG : 'N U T, 0, 0, 1',
	X =  103.000  mm,	Y =  67.000  mm,	Z =   15.000 mm,
	W =180.000 deg,	P =   0.000 deg,	R =    90.000 deg
};
P[3815]{
   GP1:
	UF : 1, UT : 1,		CONFIG : 'N U T, 0, 0, 1',
	X =  103.000  mm,	Y =  67.000  mm,	Z =   0.600 mm,
	W =180.000 deg,	P =   0.000 deg,	R =    90.000 deg
};
P[3816]{
   GP1:
	UF : 1, UT : 1,		CONFIG : 'N U T, 0, 0, 1',
	X =  103.000  mm,	Y =  67.000  mm,	Z =   15.000 mm,
	W =180.000 deg,	P =   0.000 deg,	R =    90.000 deg
};
P[3817]{
   GP1:
	UF : 1, UT : 1,		CONFIG : 'N U T, 0, 0, 1',
	X =  106.000  mm,	Y =  67.000  mm,	Z =   15.000 mm,
	W =180.000 deg,	P =   0.000 deg,	R =    90.000 deg
};
P[3818]{
   GP1:
	UF : 1, UT : 1,		CONFIG : 'N U T, 0, 0, 1',
	X =  106.000  mm,	Y =  67.000  mm,	Z =   0.600 mm,
	W =180.000 deg,	P =   0.000 deg,	R =    90.000 deg
};
P[3819]{
   GP1:
	UF : 1, UT : 1,		CONFIG : 'N U T, 0, 0, 1',
	X =  106.000  mm,	Y =  67.000  mm,	Z =   15.000 mm,
	W =180.000 deg,	P =   0.000 deg,	R =    90.000 deg
};
P[3820]{
   GP1:
	UF : 1, UT : 1,		CONFIG : 'N U T, 0, 0, 1',
	X =  109.000  mm,	Y =  67.000  mm,	Z =   15.000 mm,
	W =180.000 deg,	P =   0.000 deg,	R =    90.000 deg
};
P[3821]{
   GP1:
	UF : 1, UT : 1,		CONFIG : 'N U T, 0, 0, 1',
	X =  109.000  mm,	Y =  67.000  mm,	Z =   0.600 mm,
	W =180.000 deg,	P =   0.000 deg,	R =    90.000 deg
};
P[3822]{
   GP1:
	UF : 1, UT : 1,		CONFIG : 'N U T, 0, 0, 1',
	X =  109.000  mm,	Y =  67.000  mm,	Z =   15.000 mm,
	W =180.000 deg,	P =   0.000 deg,	R =    90.000 deg
};
P[3823]{
   GP1:
	UF : 1, UT : 1,		CONFIG : 'N U T, 0, 0, 1',
	X =  112.000  mm,	Y =  67.000  mm,	Z =   15.000 mm,
	W =180.000 deg,	P =   0.000 deg,	R =    90.000 deg
};
P[3824]{
   GP1:
	UF : 1, UT : 1,		CONFIG : 'N U T, 0, 0, 1',
	X =  112.000  mm,	Y =  67.000  mm,	Z =   0.600 mm,
	W =180.000 deg,	P =   0.000 deg,	R =    90.000 deg
};
P[3825]{
   GP1:
	UF : 1, UT : 1,		CONFIG : 'N U T, 0, 0, 1',
	X =  112.000  mm,	Y =  67.000  mm,	Z =   15.000 mm,
	W =180.000 deg,	P =   0.000 deg,	R =    90.000 deg
};
P[3826]{
   GP1:
	UF : 1, UT : 1,		CONFIG : 'N U T, 0, 0, 1',
	X =  115.000  mm,	Y =  67.000  mm,	Z =   15.000 mm,
	W =180.000 deg,	P =   0.000 deg,	R =    90.000 deg
};
P[3827]{
   GP1:
	UF : 1, UT : 1,		CONFIG : 'N U T, 0, 0, 1',
	X =  115.000  mm,	Y =  67.000  mm,	Z =   0.600 mm,
	W =180.000 deg,	P =   0.000 deg,	R =    90.000 deg
};
P[3828]{
   GP1:
	UF : 1, UT : 1,		CONFIG : 'N U T, 0, 0, 1',
	X =  115.000  mm,	Y =  67.000  mm,	Z =   15.000 mm,
	W =180.000 deg,	P =   0.000 deg,	R =    90.000 deg
};
P[3829]{
   GP1:
	UF : 1, UT : 1,		CONFIG : 'N U T, 0, 0, 1',
	X =  130.000  mm,	Y =  67.000  mm,	Z =   15.000 mm,
	W =180.000 deg,	P =   0.000 deg,	R =    90.000 deg
};
P[3830]{
   GP1:
	UF : 1, UT : 1,		CONFIG : 'N U T, 0, 0, 1',
	X =  130.000  mm,	Y =  67.000  mm,	Z =   0.600 mm,
	W =180.000 deg,	P =   0.000 deg,	R =    90.000 deg
};
P[3831]{
   GP1:
	UF : 1, UT : 1,		CONFIG : 'N U T, 0, 0, 1',
	X =  130.000  mm,	Y =  67.000  mm,	Z =   15.000 mm,
	W =180.000 deg,	P =   0.000 deg,	R =    90.000 deg
};
P[3835]{
   GP1:
	UF : 1, UT : 1,		CONFIG : 'N U T, 0, 0, 1',
	X =  136.000  mm,	Y =  67.000  mm,	Z =   15.000 mm,
	W =180.000 deg,	P =   0.000 deg,	R =    90.000 deg
};
P[3836]{
   GP1:
	UF : 1, UT : 1,		CONFIG : 'N U T, 0, 0, 1',
	X =  136.000  mm,	Y =  67.000  mm,	Z =   0.600 mm,
	W =180.000 deg,	P =   0.000 deg,	R =    90.000 deg
};
P[3837]{
   GP1:
	UF : 1, UT : 1,		CONFIG : 'N U T, 0, 0, 1',
	X =  136.000  mm,	Y =  67.000  mm,	Z =   15.000 mm,
	W =180.000 deg,	P =   0.000 deg,	R =    90.000 deg
};
P[3841]{
   GP1:
	UF : 1, UT : 1,		CONFIG : 'N U T, 0, 0, 1',
	X =  142.000  mm,	Y =  67.000  mm,	Z =   15.000 mm,
	W =180.000 deg,	P =   0.000 deg,	R =    90.000 deg
};
P[3842]{
   GP1:
	UF : 1, UT : 1,		CONFIG : 'N U T, 0, 0, 1',
	X =  142.000  mm,	Y =  67.000  mm,	Z =   0.600 mm,
	W =180.000 deg,	P =   0.000 deg,	R =    90.000 deg
};
P[3843]{
   GP1:
	UF : 1, UT : 1,		CONFIG : 'N U T, 0, 0, 1',
	X =  142.000  mm,	Y =  67.000  mm,	Z =   15.000 mm,
	W =180.000 deg,	P =   0.000 deg,	R =    90.000 deg
};
P[3844]{
   GP1:
	UF : 1, UT : 1,		CONFIG : 'N U T, 0, 0, 1',
	X =  145.000  mm,	Y =  67.000  mm,	Z =   15.000 mm,
	W =180.000 deg,	P =   0.000 deg,	R =    90.000 deg
};
P[3845]{
   GP1:
	UF : 1, UT : 1,		CONFIG : 'N U T, 0, 0, 1',
	X =  145.000  mm,	Y =  67.000  mm,	Z =   0.600 mm,
	W =180.000 deg,	P =   0.000 deg,	R =    90.000 deg
};
P[3846]{
   GP1:
	UF : 1, UT : 1,		CONFIG : 'N U T, 0, 0, 1',
	X =  145.000  mm,	Y =  67.000  mm,	Z =   15.000 mm,
	W =180.000 deg,	P =   0.000 deg,	R =    90.000 deg
};
P[3847]{
   GP1:
	UF : 1, UT : 1,		CONFIG : 'N U T, 0, 0, 1',
	X =  172.000  mm,	Y =  67.000  mm,	Z =   15.000 mm,
	W =180.000 deg,	P =   0.000 deg,	R =    90.000 deg
};
P[3848]{
   GP1:
	UF : 1, UT : 1,		CONFIG : 'N U T, 0, 0, 1',
	X =  172.000  mm,	Y =  67.000  mm,	Z =   0.600 mm,
	W =180.000 deg,	P =   0.000 deg,	R =    90.000 deg
};
P[3849]{
   GP1:
	UF : 1, UT : 1,		CONFIG : 'N U T, 0, 0, 1',
	X =  172.000  mm,	Y =  67.000  mm,	Z =   15.000 mm,
	W =180.000 deg,	P =   0.000 deg,	R =    90.000 deg
};
P[3850]{
   GP1:
	UF : 1, UT : 1,		CONFIG : 'N U T, 0, 0, 1',
	X =  175.000  mm,	Y =  67.000  mm,	Z =   15.000 mm,
	W =180.000 deg,	P =   0.000 deg,	R =    90.000 deg
};
P[3851]{
   GP1:
	UF : 1, UT : 1,		CONFIG : 'N U T, 0, 0, 1',
	X =  175.000  mm,	Y =  67.000  mm,	Z =   0.600 mm,
	W =180.000 deg,	P =   0.000 deg,	R =    90.000 deg
};
P[3852]{
   GP1:
	UF : 1, UT : 1,		CONFIG : 'N U T, 0, 0, 1',
	X =  175.000  mm,	Y =  67.000  mm,	Z =   15.000 mm,
	W =180.000 deg,	P =   0.000 deg,	R =    90.000 deg
};
P[3853]{
   GP1:
	UF : 1, UT : 1,		CONFIG : 'N U T, 0, 0, 1',
	X =  178.000  mm,	Y =  67.000  mm,	Z =   15.000 mm,
	W =180.000 deg,	P =   0.000 deg,	R =    90.000 deg
};
P[3854]{
   GP1:
	UF : 1, UT : 1,		CONFIG : 'N U T, 0, 0, 1',
	X =  178.000  mm,	Y =  67.000  mm,	Z =   0.600 mm,
	W =180.000 deg,	P =   0.000 deg,	R =    90.000 deg
};
P[3855]{
   GP1:
	UF : 1, UT : 1,		CONFIG : 'N U T, 0, 0, 1',
	X =  178.000  mm,	Y =  67.000  mm,	Z =   15.000 mm,
	W =180.000 deg,	P =   0.000 deg,	R =    90.000 deg
};
P[3856]{
   GP1:
	UF : 1, UT : 1,		CONFIG : 'N U T, 0, 0, 1',
	X =  1.000  mm,	Y =  70.000  mm,	Z =   15.000 mm,
	W =180.000 deg,	P =   0.000 deg,	R =    90.000 deg
};
P[3857]{
   GP1:
	UF : 1, UT : 1,		CONFIG : 'N U T, 0, 0, 1',
	X =  1.000  mm,	Y =  70.000  mm,	Z =   0.600 mm,
	W =180.000 deg,	P =   0.000 deg,	R =    90.000 deg
};
P[3858]{
   GP1:
	UF : 1, UT : 1,		CONFIG : 'N U T, 0, 0, 1',
	X =  1.000  mm,	Y =  70.000  mm,	Z =   15.000 mm,
	W =180.000 deg,	P =   0.000 deg,	R =    90.000 deg
};
P[3859]{
   GP1:
	UF : 1, UT : 1,		CONFIG : 'N U T, 0, 0, 1',
	X =  4.000  mm,	Y =  70.000  mm,	Z =   15.000 mm,
	W =180.000 deg,	P =   0.000 deg,	R =    90.000 deg
};
P[3860]{
   GP1:
	UF : 1, UT : 1,		CONFIG : 'N U T, 0, 0, 1',
	X =  4.000  mm,	Y =  70.000  mm,	Z =   0.600 mm,
	W =180.000 deg,	P =   0.000 deg,	R =    90.000 deg
};
P[3861]{
   GP1:
	UF : 1, UT : 1,		CONFIG : 'N U T, 0, 0, 1',
	X =  4.000  mm,	Y =  70.000  mm,	Z =   15.000 mm,
	W =180.000 deg,	P =   0.000 deg,	R =    90.000 deg
};
P[3862]{
   GP1:
	UF : 1, UT : 1,		CONFIG : 'N U T, 0, 0, 1',
	X =  7.000  mm,	Y =  70.000  mm,	Z =   15.000 mm,
	W =180.000 deg,	P =   0.000 deg,	R =    90.000 deg
};
P[3863]{
   GP1:
	UF : 1, UT : 1,		CONFIG : 'N U T, 0, 0, 1',
	X =  7.000  mm,	Y =  70.000  mm,	Z =   0.600 mm,
	W =180.000 deg,	P =   0.000 deg,	R =    90.000 deg
};
P[3864]{
   GP1:
	UF : 1, UT : 1,		CONFIG : 'N U T, 0, 0, 1',
	X =  7.000  mm,	Y =  70.000  mm,	Z =   15.000 mm,
	W =180.000 deg,	P =   0.000 deg,	R =    90.000 deg
};
P[3865]{
   GP1:
	UF : 1, UT : 1,		CONFIG : 'N U T, 0, 0, 1',
	X =  10.000  mm,	Y =  70.000  mm,	Z =   15.000 mm,
	W =180.000 deg,	P =   0.000 deg,	R =    90.000 deg
};
P[3866]{
   GP1:
	UF : 1, UT : 1,		CONFIG : 'N U T, 0, 0, 1',
	X =  10.000  mm,	Y =  70.000  mm,	Z =   0.600 mm,
	W =180.000 deg,	P =   0.000 deg,	R =    90.000 deg
};
P[3867]{
   GP1:
	UF : 1, UT : 1,		CONFIG : 'N U T, 0, 0, 1',
	X =  10.000  mm,	Y =  70.000  mm,	Z =   15.000 mm,
	W =180.000 deg,	P =   0.000 deg,	R =    90.000 deg
};
P[3868]{
   GP1:
	UF : 1, UT : 1,		CONFIG : 'N U T, 0, 0, 1',
	X =  13.000  mm,	Y =  70.000  mm,	Z =   15.000 mm,
	W =180.000 deg,	P =   0.000 deg,	R =    90.000 deg
};
P[3869]{
   GP1:
	UF : 1, UT : 1,		CONFIG : 'N U T, 0, 0, 1',
	X =  13.000  mm,	Y =  70.000  mm,	Z =   0.600 mm,
	W =180.000 deg,	P =   0.000 deg,	R =    90.000 deg
};
P[3870]{
   GP1:
	UF : 1, UT : 1,		CONFIG : 'N U T, 0, 0, 1',
	X =  13.000  mm,	Y =  70.000  mm,	Z =   15.000 mm,
	W =180.000 deg,	P =   0.000 deg,	R =    90.000 deg
};
P[3871]{
   GP1:
	UF : 1, UT : 1,		CONFIG : 'N U T, 0, 0, 1',
	X =  16.000  mm,	Y =  70.000  mm,	Z =   15.000 mm,
	W =180.000 deg,	P =   0.000 deg,	R =    90.000 deg
};
P[3872]{
   GP1:
	UF : 1, UT : 1,		CONFIG : 'N U T, 0, 0, 1',
	X =  16.000  mm,	Y =  70.000  mm,	Z =   0.600 mm,
	W =180.000 deg,	P =   0.000 deg,	R =    90.000 deg
};
P[3873]{
   GP1:
	UF : 1, UT : 1,		CONFIG : 'N U T, 0, 0, 1',
	X =  16.000  mm,	Y =  70.000  mm,	Z =   15.000 mm,
	W =180.000 deg,	P =   0.000 deg,	R =    90.000 deg
};
P[3874]{
   GP1:
	UF : 1, UT : 1,		CONFIG : 'N U T, 0, 0, 1',
	X =  19.000  mm,	Y =  70.000  mm,	Z =   15.000 mm,
	W =180.000 deg,	P =   0.000 deg,	R =    90.000 deg
};
P[3875]{
   GP1:
	UF : 1, UT : 1,		CONFIG : 'N U T, 0, 0, 1',
	X =  19.000  mm,	Y =  70.000  mm,	Z =   0.600 mm,
	W =180.000 deg,	P =   0.000 deg,	R =    90.000 deg
};
P[3876]{
   GP1:
	UF : 1, UT : 1,		CONFIG : 'N U T, 0, 0, 1',
	X =  19.000  mm,	Y =  70.000  mm,	Z =   15.000 mm,
	W =180.000 deg,	P =   0.000 deg,	R =    90.000 deg
};
P[3877]{
   GP1:
	UF : 1, UT : 1,		CONFIG : 'N U T, 0, 0, 1',
	X =  22.000  mm,	Y =  70.000  mm,	Z =   15.000 mm,
	W =180.000 deg,	P =   0.000 deg,	R =    90.000 deg
};
P[3878]{
   GP1:
	UF : 1, UT : 1,		CONFIG : 'N U T, 0, 0, 1',
	X =  22.000  mm,	Y =  70.000  mm,	Z =   0.600 mm,
	W =180.000 deg,	P =   0.000 deg,	R =    90.000 deg
};
P[3879]{
   GP1:
	UF : 1, UT : 1,		CONFIG : 'N U T, 0, 0, 1',
	X =  22.000  mm,	Y =  70.000  mm,	Z =   15.000 mm,
	W =180.000 deg,	P =   0.000 deg,	R =    90.000 deg
};
P[3880]{
   GP1:
	UF : 1, UT : 1,		CONFIG : 'N U T, 0, 0, 1',
	X =  25.000  mm,	Y =  70.000  mm,	Z =   15.000 mm,
	W =180.000 deg,	P =   0.000 deg,	R =    90.000 deg
};
P[3881]{
   GP1:
	UF : 1, UT : 1,		CONFIG : 'N U T, 0, 0, 1',
	X =  25.000  mm,	Y =  70.000  mm,	Z =   0.600 mm,
	W =180.000 deg,	P =   0.000 deg,	R =    90.000 deg
};
P[3882]{
   GP1:
	UF : 1, UT : 1,		CONFIG : 'N U T, 0, 0, 1',
	X =  25.000  mm,	Y =  70.000  mm,	Z =   15.000 mm,
	W =180.000 deg,	P =   0.000 deg,	R =    90.000 deg
};
P[3883]{
   GP1:
	UF : 1, UT : 1,		CONFIG : 'N U T, 0, 0, 1',
	X =  28.000  mm,	Y =  70.000  mm,	Z =   15.000 mm,
	W =180.000 deg,	P =   0.000 deg,	R =    90.000 deg
};
P[3884]{
   GP1:
	UF : 1, UT : 1,		CONFIG : 'N U T, 0, 0, 1',
	X =  28.000  mm,	Y =  70.000  mm,	Z =   0.600 mm,
	W =180.000 deg,	P =   0.000 deg,	R =    90.000 deg
};
P[3885]{
   GP1:
	UF : 1, UT : 1,		CONFIG : 'N U T, 0, 0, 1',
	X =  28.000  mm,	Y =  70.000  mm,	Z =   15.000 mm,
	W =180.000 deg,	P =   0.000 deg,	R =    90.000 deg
};
P[3886]{
   GP1:
	UF : 1, UT : 1,		CONFIG : 'N U T, 0, 0, 1',
	X =  34.000  mm,	Y =  70.000  mm,	Z =   15.000 mm,
	W =180.000 deg,	P =   0.000 deg,	R =    90.000 deg
};
P[3887]{
   GP1:
	UF : 1, UT : 1,		CONFIG : 'N U T, 0, 0, 1',
	X =  34.000  mm,	Y =  70.000  mm,	Z =   0.600 mm,
	W =180.000 deg,	P =   0.000 deg,	R =    90.000 deg
};
P[3888]{
   GP1:
	UF : 1, UT : 1,		CONFIG : 'N U T, 0, 0, 1',
	X =  34.000  mm,	Y =  70.000  mm,	Z =   15.000 mm,
	W =180.000 deg,	P =   0.000 deg,	R =    90.000 deg
};
P[3889]{
   GP1:
	UF : 1, UT : 1,		CONFIG : 'N U T, 0, 0, 1',
	X =  37.000  mm,	Y =  70.000  mm,	Z =   15.000 mm,
	W =180.000 deg,	P =   0.000 deg,	R =    90.000 deg
};
P[3890]{
   GP1:
	UF : 1, UT : 1,		CONFIG : 'N U T, 0, 0, 1',
	X =  37.000  mm,	Y =  70.000  mm,	Z =   0.600 mm,
	W =180.000 deg,	P =   0.000 deg,	R =    90.000 deg
};
P[3891]{
   GP1:
	UF : 1, UT : 1,		CONFIG : 'N U T, 0, 0, 1',
	X =  37.000  mm,	Y =  70.000  mm,	Z =   15.000 mm,
	W =180.000 deg,	P =   0.000 deg,	R =    90.000 deg
};
P[3892]{
   GP1:
	UF : 1, UT : 1,		CONFIG : 'N U T, 0, 0, 1',
	X =  40.000  mm,	Y =  70.000  mm,	Z =   15.000 mm,
	W =180.000 deg,	P =   0.000 deg,	R =    90.000 deg
};
P[3893]{
   GP1:
	UF : 1, UT : 1,		CONFIG : 'N U T, 0, 0, 1',
	X =  40.000  mm,	Y =  70.000  mm,	Z =   0.600 mm,
	W =180.000 deg,	P =   0.000 deg,	R =    90.000 deg
};
P[3894]{
   GP1:
	UF : 1, UT : 1,		CONFIG : 'N U T, 0, 0, 1',
	X =  40.000  mm,	Y =  70.000  mm,	Z =   15.000 mm,
	W =180.000 deg,	P =   0.000 deg,	R =    90.000 deg
};
P[3895]{
   GP1:
	UF : 1, UT : 1,		CONFIG : 'N U T, 0, 0, 1',
	X =  43.000  mm,	Y =  70.000  mm,	Z =   15.000 mm,
	W =180.000 deg,	P =   0.000 deg,	R =    90.000 deg
};
P[3896]{
   GP1:
	UF : 1, UT : 1,		CONFIG : 'N U T, 0, 0, 1',
	X =  43.000  mm,	Y =  70.000  mm,	Z =   0.600 mm,
	W =180.000 deg,	P =   0.000 deg,	R =    90.000 deg
};
P[3897]{
   GP1:
	UF : 1, UT : 1,		CONFIG : 'N U T, 0, 0, 1',
	X =  43.000  mm,	Y =  70.000  mm,	Z =   15.000 mm,
	W =180.000 deg,	P =   0.000 deg,	R =    90.000 deg
};
P[3898]{
   GP1:
	UF : 1, UT : 1,		CONFIG : 'N U T, 0, 0, 1',
	X =  46.000  mm,	Y =  70.000  mm,	Z =   15.000 mm,
	W =180.000 deg,	P =   0.000 deg,	R =    90.000 deg
};
P[3899]{
   GP1:
	UF : 1, UT : 1,		CONFIG : 'N U T, 0, 0, 1',
	X =  46.000  mm,	Y =  70.000  mm,	Z =   0.600 mm,
	W =180.000 deg,	P =   0.000 deg,	R =    90.000 deg
};
P[3900]{
   GP1:
	UF : 1, UT : 1,		CONFIG : 'N U T, 0, 0, 1',
	X =  46.000  mm,	Y =  70.000  mm,	Z =   15.000 mm,
	W =180.000 deg,	P =   0.000 deg,	R =    90.000 deg
};
P[3901]{
   GP1:
	UF : 1, UT : 1,		CONFIG : 'N U T, 0, 0, 1',
	X =  49.000  mm,	Y =  70.000  mm,	Z =   15.000 mm,
	W =180.000 deg,	P =   0.000 deg,	R =    90.000 deg
};
P[3902]{
   GP1:
	UF : 1, UT : 1,		CONFIG : 'N U T, 0, 0, 1',
	X =  49.000  mm,	Y =  70.000  mm,	Z =   0.600 mm,
	W =180.000 deg,	P =   0.000 deg,	R =    90.000 deg
};
P[3903]{
   GP1:
	UF : 1, UT : 1,		CONFIG : 'N U T, 0, 0, 1',
	X =  49.000  mm,	Y =  70.000  mm,	Z =   15.000 mm,
	W =180.000 deg,	P =   0.000 deg,	R =    90.000 deg
};
P[3904]{
   GP1:
	UF : 1, UT : 1,		CONFIG : 'N U T, 0, 0, 1',
	X =  52.000  mm,	Y =  70.000  mm,	Z =   15.000 mm,
	W =180.000 deg,	P =   0.000 deg,	R =    90.000 deg
};
P[3905]{
   GP1:
	UF : 1, UT : 1,		CONFIG : 'N U T, 0, 0, 1',
	X =  52.000  mm,	Y =  70.000  mm,	Z =   0.600 mm,
	W =180.000 deg,	P =   0.000 deg,	R =    90.000 deg
};
P[3906]{
   GP1:
	UF : 1, UT : 1,		CONFIG : 'N U T, 0, 0, 1',
	X =  52.000  mm,	Y =  70.000  mm,	Z =   15.000 mm,
	W =180.000 deg,	P =   0.000 deg,	R =    90.000 deg
};
P[3907]{
   GP1:
	UF : 1, UT : 1,		CONFIG : 'N U T, 0, 0, 1',
	X =  55.000  mm,	Y =  70.000  mm,	Z =   15.000 mm,
	W =180.000 deg,	P =   0.000 deg,	R =    90.000 deg
};
P[3908]{
   GP1:
	UF : 1, UT : 1,		CONFIG : 'N U T, 0, 0, 1',
	X =  55.000  mm,	Y =  70.000  mm,	Z =   0.600 mm,
	W =180.000 deg,	P =   0.000 deg,	R =    90.000 deg
};
P[3909]{
   GP1:
	UF : 1, UT : 1,		CONFIG : 'N U T, 0, 0, 1',
	X =  55.000  mm,	Y =  70.000  mm,	Z =   15.000 mm,
	W =180.000 deg,	P =   0.000 deg,	R =    90.000 deg
};
P[3910]{
   GP1:
	UF : 1, UT : 1,		CONFIG : 'N U T, 0, 0, 1',
	X =  58.000  mm,	Y =  70.000  mm,	Z =   15.000 mm,
	W =180.000 deg,	P =   0.000 deg,	R =    90.000 deg
};
P[3911]{
   GP1:
	UF : 1, UT : 1,		CONFIG : 'N U T, 0, 0, 1',
	X =  58.000  mm,	Y =  70.000  mm,	Z =   0.600 mm,
	W =180.000 deg,	P =   0.000 deg,	R =    90.000 deg
};
P[3912]{
   GP1:
	UF : 1, UT : 1,		CONFIG : 'N U T, 0, 0, 1',
	X =  58.000  mm,	Y =  70.000  mm,	Z =   15.000 mm,
	W =180.000 deg,	P =   0.000 deg,	R =    90.000 deg
};
P[3913]{
   GP1:
	UF : 1, UT : 1,		CONFIG : 'N U T, 0, 0, 1',
	X =  61.000  mm,	Y =  70.000  mm,	Z =   15.000 mm,
	W =180.000 deg,	P =   0.000 deg,	R =    90.000 deg
};
P[3914]{
   GP1:
	UF : 1, UT : 1,		CONFIG : 'N U T, 0, 0, 1',
	X =  61.000  mm,	Y =  70.000  mm,	Z =   0.600 mm,
	W =180.000 deg,	P =   0.000 deg,	R =    90.000 deg
};
P[3915]{
   GP1:
	UF : 1, UT : 1,		CONFIG : 'N U T, 0, 0, 1',
	X =  61.000  mm,	Y =  70.000  mm,	Z =   15.000 mm,
	W =180.000 deg,	P =   0.000 deg,	R =    90.000 deg
};
P[3916]{
   GP1:
	UF : 1, UT : 1,		CONFIG : 'N U T, 0, 0, 1',
	X =  64.000  mm,	Y =  70.000  mm,	Z =   15.000 mm,
	W =180.000 deg,	P =   0.000 deg,	R =    90.000 deg
};
P[3917]{
   GP1:
	UF : 1, UT : 1,		CONFIG : 'N U T, 0, 0, 1',
	X =  64.000  mm,	Y =  70.000  mm,	Z =   0.600 mm,
	W =180.000 deg,	P =   0.000 deg,	R =    90.000 deg
};
P[3918]{
   GP1:
	UF : 1, UT : 1,		CONFIG : 'N U T, 0, 0, 1',
	X =  64.000  mm,	Y =  70.000  mm,	Z =   15.000 mm,
	W =180.000 deg,	P =   0.000 deg,	R =    90.000 deg
};
P[3919]{
   GP1:
	UF : 1, UT : 1,		CONFIG : 'N U T, 0, 0, 1',
	X =  67.000  mm,	Y =  70.000  mm,	Z =   15.000 mm,
	W =180.000 deg,	P =   0.000 deg,	R =    90.000 deg
};
P[3920]{
   GP1:
	UF : 1, UT : 1,		CONFIG : 'N U T, 0, 0, 1',
	X =  67.000  mm,	Y =  70.000  mm,	Z =   0.600 mm,
	W =180.000 deg,	P =   0.000 deg,	R =    90.000 deg
};
P[3921]{
   GP1:
	UF : 1, UT : 1,		CONFIG : 'N U T, 0, 0, 1',
	X =  67.000  mm,	Y =  70.000  mm,	Z =   15.000 mm,
	W =180.000 deg,	P =   0.000 deg,	R =    90.000 deg
};
P[3922]{
   GP1:
	UF : 1, UT : 1,		CONFIG : 'N U T, 0, 0, 1',
	X =  70.000  mm,	Y =  70.000  mm,	Z =   15.000 mm,
	W =180.000 deg,	P =   0.000 deg,	R =    90.000 deg
};
P[3923]{
   GP1:
	UF : 1, UT : 1,		CONFIG : 'N U T, 0, 0, 1',
	X =  70.000  mm,	Y =  70.000  mm,	Z =   0.600 mm,
	W =180.000 deg,	P =   0.000 deg,	R =    90.000 deg
};
P[3924]{
   GP1:
	UF : 1, UT : 1,		CONFIG : 'N U T, 0, 0, 1',
	X =  70.000  mm,	Y =  70.000  mm,	Z =   15.000 mm,
	W =180.000 deg,	P =   0.000 deg,	R =    90.000 deg
};
P[3928]{
   GP1:
	UF : 1, UT : 1,		CONFIG : 'N U T, 0, 0, 1',
	X =  76.000  mm,	Y =  70.000  mm,	Z =   15.000 mm,
	W =180.000 deg,	P =   0.000 deg,	R =    90.000 deg
};
P[3929]{
   GP1:
	UF : 1, UT : 1,		CONFIG : 'N U T, 0, 0, 1',
	X =  76.000  mm,	Y =  70.000  mm,	Z =   0.600 mm,
	W =180.000 deg,	P =   0.000 deg,	R =    90.000 deg
};
P[3930]{
   GP1:
	UF : 1, UT : 1,		CONFIG : 'N U T, 0, 0, 1',
	X =  76.000  mm,	Y =  70.000  mm,	Z =   15.000 mm,
	W =180.000 deg,	P =   0.000 deg,	R =    90.000 deg
};
P[3931]{
   GP1:
	UF : 1, UT : 1,		CONFIG : 'N U T, 0, 0, 1',
	X =  79.000  mm,	Y =  70.000  mm,	Z =   15.000 mm,
	W =180.000 deg,	P =   0.000 deg,	R =    90.000 deg
};
P[3932]{
   GP1:
	UF : 1, UT : 1,		CONFIG : 'N U T, 0, 0, 1',
	X =  79.000  mm,	Y =  70.000  mm,	Z =   0.600 mm,
	W =180.000 deg,	P =   0.000 deg,	R =    90.000 deg
};
P[3933]{
   GP1:
	UF : 1, UT : 1,		CONFIG : 'N U T, 0, 0, 1',
	X =  79.000  mm,	Y =  70.000  mm,	Z =   15.000 mm,
	W =180.000 deg,	P =   0.000 deg,	R =    90.000 deg
};
P[3934]{
   GP1:
	UF : 1, UT : 1,		CONFIG : 'N U T, 0, 0, 1',
	X =  82.000  mm,	Y =  70.000  mm,	Z =   15.000 mm,
	W =180.000 deg,	P =   0.000 deg,	R =    90.000 deg
};
P[3935]{
   GP1:
	UF : 1, UT : 1,		CONFIG : 'N U T, 0, 0, 1',
	X =  82.000  mm,	Y =  70.000  mm,	Z =   0.600 mm,
	W =180.000 deg,	P =   0.000 deg,	R =    90.000 deg
};
P[3936]{
   GP1:
	UF : 1, UT : 1,		CONFIG : 'N U T, 0, 0, 1',
	X =  82.000  mm,	Y =  70.000  mm,	Z =   15.000 mm,
	W =180.000 deg,	P =   0.000 deg,	R =    90.000 deg
};
P[3937]{
   GP1:
	UF : 1, UT : 1,		CONFIG : 'N U T, 0, 0, 1',
	X =  85.000  mm,	Y =  70.000  mm,	Z =   15.000 mm,
	W =180.000 deg,	P =   0.000 deg,	R =    90.000 deg
};
P[3938]{
   GP1:
	UF : 1, UT : 1,		CONFIG : 'N U T, 0, 0, 1',
	X =  85.000  mm,	Y =  70.000  mm,	Z =   0.600 mm,
	W =180.000 deg,	P =   0.000 deg,	R =    90.000 deg
};
P[3939]{
   GP1:
	UF : 1, UT : 1,		CONFIG : 'N U T, 0, 0, 1',
	X =  85.000  mm,	Y =  70.000  mm,	Z =   15.000 mm,
	W =180.000 deg,	P =   0.000 deg,	R =    90.000 deg
};
P[3940]{
   GP1:
	UF : 1, UT : 1,		CONFIG : 'N U T, 0, 0, 1',
	X =  88.000  mm,	Y =  70.000  mm,	Z =   15.000 mm,
	W =180.000 deg,	P =   0.000 deg,	R =    90.000 deg
};
P[3941]{
   GP1:
	UF : 1, UT : 1,		CONFIG : 'N U T, 0, 0, 1',
	X =  88.000  mm,	Y =  70.000  mm,	Z =   0.600 mm,
	W =180.000 deg,	P =   0.000 deg,	R =    90.000 deg
};
P[3942]{
   GP1:
	UF : 1, UT : 1,		CONFIG : 'N U T, 0, 0, 1',
	X =  88.000  mm,	Y =  70.000  mm,	Z =   15.000 mm,
	W =180.000 deg,	P =   0.000 deg,	R =    90.000 deg
};
P[3943]{
   GP1:
	UF : 1, UT : 1,		CONFIG : 'N U T, 0, 0, 1',
	X =  91.000  mm,	Y =  70.000  mm,	Z =   15.000 mm,
	W =180.000 deg,	P =   0.000 deg,	R =    90.000 deg
};
P[3944]{
   GP1:
	UF : 1, UT : 1,		CONFIG : 'N U T, 0, 0, 1',
	X =  91.000  mm,	Y =  70.000  mm,	Z =   0.600 mm,
	W =180.000 deg,	P =   0.000 deg,	R =    90.000 deg
};
P[3945]{
   GP1:
	UF : 1, UT : 1,		CONFIG : 'N U T, 0, 0, 1',
	X =  91.000  mm,	Y =  70.000  mm,	Z =   15.000 mm,
	W =180.000 deg,	P =   0.000 deg,	R =    90.000 deg
};
P[3946]{
   GP1:
	UF : 1, UT : 1,		CONFIG : 'N U T, 0, 0, 1',
	X =  94.000  mm,	Y =  70.000  mm,	Z =   15.000 mm,
	W =180.000 deg,	P =   0.000 deg,	R =    90.000 deg
};
P[3947]{
   GP1:
	UF : 1, UT : 1,		CONFIG : 'N U T, 0, 0, 1',
	X =  94.000  mm,	Y =  70.000  mm,	Z =   0.600 mm,
	W =180.000 deg,	P =   0.000 deg,	R =    90.000 deg
};
P[3948]{
   GP1:
	UF : 1, UT : 1,		CONFIG : 'N U T, 0, 0, 1',
	X =  94.000  mm,	Y =  70.000  mm,	Z =   15.000 mm,
	W =180.000 deg,	P =   0.000 deg,	R =    90.000 deg
};
P[3949]{
   GP1:
	UF : 1, UT : 1,		CONFIG : 'N U T, 0, 0, 1',
	X =  97.000  mm,	Y =  70.000  mm,	Z =   15.000 mm,
	W =180.000 deg,	P =   0.000 deg,	R =    90.000 deg
};
P[3950]{
   GP1:
	UF : 1, UT : 1,		CONFIG : 'N U T, 0, 0, 1',
	X =  97.000  mm,	Y =  70.000  mm,	Z =   0.600 mm,
	W =180.000 deg,	P =   0.000 deg,	R =    90.000 deg
};
P[3951]{
   GP1:
	UF : 1, UT : 1,		CONFIG : 'N U T, 0, 0, 1',
	X =  97.000  mm,	Y =  70.000  mm,	Z =   15.000 mm,
	W =180.000 deg,	P =   0.000 deg,	R =    90.000 deg
};
P[3952]{
   GP1:
	UF : 1, UT : 1,		CONFIG : 'N U T, 0, 0, 1',
	X =  100.000  mm,	Y =  70.000  mm,	Z =   15.000 mm,
	W =180.000 deg,	P =   0.000 deg,	R =    90.000 deg
};
P[3953]{
   GP1:
	UF : 1, UT : 1,		CONFIG : 'N U T, 0, 0, 1',
	X =  100.000  mm,	Y =  70.000  mm,	Z =   0.600 mm,
	W =180.000 deg,	P =   0.000 deg,	R =    90.000 deg
};
P[3954]{
   GP1:
	UF : 1, UT : 1,		CONFIG : 'N U T, 0, 0, 1',
	X =  100.000  mm,	Y =  70.000  mm,	Z =   15.000 mm,
	W =180.000 deg,	P =   0.000 deg,	R =    90.000 deg
};
P[3955]{
   GP1:
	UF : 1, UT : 1,		CONFIG : 'N U T, 0, 0, 1',
	X =  103.000  mm,	Y =  70.000  mm,	Z =   15.000 mm,
	W =180.000 deg,	P =   0.000 deg,	R =    90.000 deg
};
P[3956]{
   GP1:
	UF : 1, UT : 1,		CONFIG : 'N U T, 0, 0, 1',
	X =  103.000  mm,	Y =  70.000  mm,	Z =   0.600 mm,
	W =180.000 deg,	P =   0.000 deg,	R =    90.000 deg
};
P[3957]{
   GP1:
	UF : 1, UT : 1,		CONFIG : 'N U T, 0, 0, 1',
	X =  103.000  mm,	Y =  70.000  mm,	Z =   15.000 mm,
	W =180.000 deg,	P =   0.000 deg,	R =    90.000 deg
};
P[3958]{
   GP1:
	UF : 1, UT : 1,		CONFIG : 'N U T, 0, 0, 1',
	X =  106.000  mm,	Y =  70.000  mm,	Z =   15.000 mm,
	W =180.000 deg,	P =   0.000 deg,	R =    90.000 deg
};
P[3959]{
   GP1:
	UF : 1, UT : 1,		CONFIG : 'N U T, 0, 0, 1',
	X =  106.000  mm,	Y =  70.000  mm,	Z =   0.600 mm,
	W =180.000 deg,	P =   0.000 deg,	R =    90.000 deg
};
P[3960]{
   GP1:
	UF : 1, UT : 1,		CONFIG : 'N U T, 0, 0, 1',
	X =  106.000  mm,	Y =  70.000  mm,	Z =   15.000 mm,
	W =180.000 deg,	P =   0.000 deg,	R =    90.000 deg
};
P[3961]{
   GP1:
	UF : 1, UT : 1,		CONFIG : 'N U T, 0, 0, 1',
	X =  109.000  mm,	Y =  70.000  mm,	Z =   15.000 mm,
	W =180.000 deg,	P =   0.000 deg,	R =    90.000 deg
};
P[3962]{
   GP1:
	UF : 1, UT : 1,		CONFIG : 'N U T, 0, 0, 1',
	X =  109.000  mm,	Y =  70.000  mm,	Z =   0.600 mm,
	W =180.000 deg,	P =   0.000 deg,	R =    90.000 deg
};
P[3963]{
   GP1:
	UF : 1, UT : 1,		CONFIG : 'N U T, 0, 0, 1',
	X =  109.000  mm,	Y =  70.000  mm,	Z =   15.000 mm,
	W =180.000 deg,	P =   0.000 deg,	R =    90.000 deg
};
P[3964]{
   GP1:
	UF : 1, UT : 1,		CONFIG : 'N U T, 0, 0, 1',
	X =  112.000  mm,	Y =  70.000  mm,	Z =   15.000 mm,
	W =180.000 deg,	P =   0.000 deg,	R =    90.000 deg
};
P[3965]{
   GP1:
	UF : 1, UT : 1,		CONFIG : 'N U T, 0, 0, 1',
	X =  112.000  mm,	Y =  70.000  mm,	Z =   0.600 mm,
	W =180.000 deg,	P =   0.000 deg,	R =    90.000 deg
};
P[3966]{
   GP1:
	UF : 1, UT : 1,		CONFIG : 'N U T, 0, 0, 1',
	X =  112.000  mm,	Y =  70.000  mm,	Z =   15.000 mm,
	W =180.000 deg,	P =   0.000 deg,	R =    90.000 deg
};
P[3967]{
   GP1:
	UF : 1, UT : 1,		CONFIG : 'N U T, 0, 0, 1',
	X =  115.000  mm,	Y =  70.000  mm,	Z =   15.000 mm,
	W =180.000 deg,	P =   0.000 deg,	R =    90.000 deg
};
P[3968]{
   GP1:
	UF : 1, UT : 1,		CONFIG : 'N U T, 0, 0, 1',
	X =  115.000  mm,	Y =  70.000  mm,	Z =   0.600 mm,
	W =180.000 deg,	P =   0.000 deg,	R =    90.000 deg
};
P[3969]{
   GP1:
	UF : 1, UT : 1,		CONFIG : 'N U T, 0, 0, 1',
	X =  115.000  mm,	Y =  70.000  mm,	Z =   15.000 mm,
	W =180.000 deg,	P =   0.000 deg,	R =    90.000 deg
};
P[3970]{
   GP1:
	UF : 1, UT : 1,		CONFIG : 'N U T, 0, 0, 1',
	X =  133.000  mm,	Y =  70.000  mm,	Z =   15.000 mm,
	W =180.000 deg,	P =   0.000 deg,	R =    90.000 deg
};
P[3971]{
   GP1:
	UF : 1, UT : 1,		CONFIG : 'N U T, 0, 0, 1',
	X =  133.000  mm,	Y =  70.000  mm,	Z =   0.600 mm,
	W =180.000 deg,	P =   0.000 deg,	R =    90.000 deg
};
P[3972]{
   GP1:
	UF : 1, UT : 1,		CONFIG : 'N U T, 0, 0, 1',
	X =  133.000  mm,	Y =  70.000  mm,	Z =   15.000 mm,
	W =180.000 deg,	P =   0.000 deg,	R =    90.000 deg
};
P[3976]{
   GP1:
	UF : 1, UT : 1,		CONFIG : 'N U T, 0, 0, 1',
	X =  139.000  mm,	Y =  70.000  mm,	Z =   15.000 mm,
	W =180.000 deg,	P =   0.000 deg,	R =    90.000 deg
};
P[3977]{
   GP1:
	UF : 1, UT : 1,		CONFIG : 'N U T, 0, 0, 1',
	X =  139.000  mm,	Y =  70.000  mm,	Z =   0.600 mm,
	W =180.000 deg,	P =   0.000 deg,	R =    90.000 deg
};
P[3978]{
   GP1:
	UF : 1, UT : 1,		CONFIG : 'N U T, 0, 0, 1',
	X =  139.000  mm,	Y =  70.000  mm,	Z =   15.000 mm,
	W =180.000 deg,	P =   0.000 deg,	R =    90.000 deg
};
P[3982]{
   GP1:
	UF : 1, UT : 1,		CONFIG : 'N U T, 0, 0, 1',
	X =  145.000  mm,	Y =  70.000  mm,	Z =   15.000 mm,
	W =180.000 deg,	P =   0.000 deg,	R =    90.000 deg
};
P[3983]{
   GP1:
	UF : 1, UT : 1,		CONFIG : 'N U T, 0, 0, 1',
	X =  145.000  mm,	Y =  70.000  mm,	Z =   0.600 mm,
	W =180.000 deg,	P =   0.000 deg,	R =    90.000 deg
};
P[3984]{
   GP1:
	UF : 1, UT : 1,		CONFIG : 'N U T, 0, 0, 1',
	X =  145.000  mm,	Y =  70.000  mm,	Z =   15.000 mm,
	W =180.000 deg,	P =   0.000 deg,	R =    90.000 deg
};
P[3988]{
   GP1:
	UF : 1, UT : 1,		CONFIG : 'N U T, 0, 0, 1',
	X =  172.000  mm,	Y =  70.000  mm,	Z =   15.000 mm,
	W =180.000 deg,	P =   0.000 deg,	R =    90.000 deg
};
P[3989]{
   GP1:
	UF : 1, UT : 1,		CONFIG : 'N U T, 0, 0, 1',
	X =  172.000  mm,	Y =  70.000  mm,	Z =   0.600 mm,
	W =180.000 deg,	P =   0.000 deg,	R =    90.000 deg
};
P[3990]{
   GP1:
	UF : 1, UT : 1,		CONFIG : 'N U T, 0, 0, 1',
	X =  172.000  mm,	Y =  70.000  mm,	Z =   15.000 mm,
	W =180.000 deg,	P =   0.000 deg,	R =    90.000 deg
};
P[3991]{
   GP1:
	UF : 1, UT : 1,		CONFIG : 'N U T, 0, 0, 1',
	X =  175.000  mm,	Y =  70.000  mm,	Z =   15.000 mm,
	W =180.000 deg,	P =   0.000 deg,	R =    90.000 deg
};
P[3992]{
   GP1:
	UF : 1, UT : 1,		CONFIG : 'N U T, 0, 0, 1',
	X =  175.000  mm,	Y =  70.000  mm,	Z =   0.600 mm,
	W =180.000 deg,	P =   0.000 deg,	R =    90.000 deg
};
P[3993]{
   GP1:
	UF : 1, UT : 1,		CONFIG : 'N U T, 0, 0, 1',
	X =  175.000  mm,	Y =  70.000  mm,	Z =   15.000 mm,
	W =180.000 deg,	P =   0.000 deg,	R =    90.000 deg
};
P[3994]{
   GP1:
	UF : 1, UT : 1,		CONFIG : 'N U T, 0, 0, 1',
	X =  178.000  mm,	Y =  70.000  mm,	Z =   15.000 mm,
	W =180.000 deg,	P =   0.000 deg,	R =    90.000 deg
};
P[3995]{
   GP1:
	UF : 1, UT : 1,		CONFIG : 'N U T, 0, 0, 1',
	X =  178.000  mm,	Y =  70.000  mm,	Z =   0.600 mm,
	W =180.000 deg,	P =   0.000 deg,	R =    90.000 deg
};
P[3996]{
   GP1:
	UF : 1, UT : 1,		CONFIG : 'N U T, 0, 0, 1',
	X =  178.000  mm,	Y =  70.000  mm,	Z =   15.000 mm,
	W =180.000 deg,	P =   0.000 deg,	R =    90.000 deg
};
P[3997]{
   GP1:
	UF : 1, UT : 1,		CONFIG : 'N U T, 0, 0, 1',
	X =  1.000  mm,	Y =  73.000  mm,	Z =   15.000 mm,
	W =180.000 deg,	P =   0.000 deg,	R =    90.000 deg
};
P[3998]{
   GP1:
	UF : 1, UT : 1,		CONFIG : 'N U T, 0, 0, 1',
	X =  1.000  mm,	Y =  73.000  mm,	Z =   0.600 mm,
	W =180.000 deg,	P =   0.000 deg,	R =    90.000 deg
};
P[3999]{
   GP1:
	UF : 1, UT : 1,		CONFIG : 'N U T, 0, 0, 1',
	X =  1.000  mm,	Y =  73.000  mm,	Z =   15.000 mm,
	W =180.000 deg,	P =   0.000 deg,	R =    90.000 deg
};
P[4000]{
   GP1:
	UF : 1, UT : 1,		CONFIG : 'N U T, 0, 0, 1',
	X =  4.000  mm,	Y =  73.000  mm,	Z =   15.000 mm,
	W =180.000 deg,	P =   0.000 deg,	R =    90.000 deg
};
P[4001]{
   GP1:
	UF : 1, UT : 1,		CONFIG : 'N U T, 0, 0, 1',
	X =  4.000  mm,	Y =  73.000  mm,	Z =   0.600 mm,
	W =180.000 deg,	P =   0.000 deg,	R =    90.000 deg
};
P[4002]{
   GP1:
	UF : 1, UT : 1,		CONFIG : 'N U T, 0, 0, 1',
	X =  4.000  mm,	Y =  73.000  mm,	Z =   15.000 mm,
	W =180.000 deg,	P =   0.000 deg,	R =    90.000 deg
};
P[4003]{
   GP1:
	UF : 1, UT : 1,		CONFIG : 'N U T, 0, 0, 1',
	X =  7.000  mm,	Y =  73.000  mm,	Z =   15.000 mm,
	W =180.000 deg,	P =   0.000 deg,	R =    90.000 deg
};
P[4004]{
   GP1:
	UF : 1, UT : 1,		CONFIG : 'N U T, 0, 0, 1',
	X =  7.000  mm,	Y =  73.000  mm,	Z =   0.600 mm,
	W =180.000 deg,	P =   0.000 deg,	R =    90.000 deg
};
P[4005]{
   GP1:
	UF : 1, UT : 1,		CONFIG : 'N U T, 0, 0, 1',
	X =  7.000  mm,	Y =  73.000  mm,	Z =   15.000 mm,
	W =180.000 deg,	P =   0.000 deg,	R =    90.000 deg
};
P[4006]{
   GP1:
	UF : 1, UT : 1,		CONFIG : 'N U T, 0, 0, 1',
	X =  10.000  mm,	Y =  73.000  mm,	Z =   15.000 mm,
	W =180.000 deg,	P =   0.000 deg,	R =    90.000 deg
};
P[4007]{
   GP1:
	UF : 1, UT : 1,		CONFIG : 'N U T, 0, 0, 1',
	X =  10.000  mm,	Y =  73.000  mm,	Z =   0.600 mm,
	W =180.000 deg,	P =   0.000 deg,	R =    90.000 deg
};
P[4008]{
   GP1:
	UF : 1, UT : 1,		CONFIG : 'N U T, 0, 0, 1',
	X =  10.000  mm,	Y =  73.000  mm,	Z =   15.000 mm,
	W =180.000 deg,	P =   0.000 deg,	R =    90.000 deg
};
P[4012]{
   GP1:
	UF : 1, UT : 1,		CONFIG : 'N U T, 0, 0, 1',
	X =  16.000  mm,	Y =  73.000  mm,	Z =   15.000 mm,
	W =180.000 deg,	P =   0.000 deg,	R =    90.000 deg
};
P[4013]{
   GP1:
	UF : 1, UT : 1,		CONFIG : 'N U T, 0, 0, 1',
	X =  16.000  mm,	Y =  73.000  mm,	Z =   0.600 mm,
	W =180.000 deg,	P =   0.000 deg,	R =    90.000 deg
};
P[4014]{
   GP1:
	UF : 1, UT : 1,		CONFIG : 'N U T, 0, 0, 1',
	X =  16.000  mm,	Y =  73.000  mm,	Z =   15.000 mm,
	W =180.000 deg,	P =   0.000 deg,	R =    90.000 deg
};
P[4015]{
   GP1:
	UF : 1, UT : 1,		CONFIG : 'N U T, 0, 0, 1',
	X =  19.000  mm,	Y =  73.000  mm,	Z =   15.000 mm,
	W =180.000 deg,	P =   0.000 deg,	R =    90.000 deg
};
P[4016]{
   GP1:
	UF : 1, UT : 1,		CONFIG : 'N U T, 0, 0, 1',
	X =  19.000  mm,	Y =  73.000  mm,	Z =   0.600 mm,
	W =180.000 deg,	P =   0.000 deg,	R =    90.000 deg
};
P[4017]{
   GP1:
	UF : 1, UT : 1,		CONFIG : 'N U T, 0, 0, 1',
	X =  19.000  mm,	Y =  73.000  mm,	Z =   15.000 mm,
	W =180.000 deg,	P =   0.000 deg,	R =    90.000 deg
};
P[4018]{
   GP1:
	UF : 1, UT : 1,		CONFIG : 'N U T, 0, 0, 1',
	X =  22.000  mm,	Y =  73.000  mm,	Z =   15.000 mm,
	W =180.000 deg,	P =   0.000 deg,	R =    90.000 deg
};
P[4019]{
   GP1:
	UF : 1, UT : 1,		CONFIG : 'N U T, 0, 0, 1',
	X =  22.000  mm,	Y =  73.000  mm,	Z =   0.600 mm,
	W =180.000 deg,	P =   0.000 deg,	R =    90.000 deg
};
P[4020]{
   GP1:
	UF : 1, UT : 1,		CONFIG : 'N U T, 0, 0, 1',
	X =  22.000  mm,	Y =  73.000  mm,	Z =   15.000 mm,
	W =180.000 deg,	P =   0.000 deg,	R =    90.000 deg
};
P[4021]{
   GP1:
	UF : 1, UT : 1,		CONFIG : 'N U T, 0, 0, 1',
	X =  25.000  mm,	Y =  73.000  mm,	Z =   15.000 mm,
	W =180.000 deg,	P =   0.000 deg,	R =    90.000 deg
};
P[4022]{
   GP1:
	UF : 1, UT : 1,		CONFIG : 'N U T, 0, 0, 1',
	X =  25.000  mm,	Y =  73.000  mm,	Z =   0.600 mm,
	W =180.000 deg,	P =   0.000 deg,	R =    90.000 deg
};
P[4023]{
   GP1:
	UF : 1, UT : 1,		CONFIG : 'N U T, 0, 0, 1',
	X =  25.000  mm,	Y =  73.000  mm,	Z =   15.000 mm,
	W =180.000 deg,	P =   0.000 deg,	R =    90.000 deg
};
P[4024]{
   GP1:
	UF : 1, UT : 1,		CONFIG : 'N U T, 0, 0, 1',
	X =  28.000  mm,	Y =  73.000  mm,	Z =   15.000 mm,
	W =180.000 deg,	P =   0.000 deg,	R =    90.000 deg
};
P[4025]{
   GP1:
	UF : 1, UT : 1,		CONFIG : 'N U T, 0, 0, 1',
	X =  28.000  mm,	Y =  73.000  mm,	Z =   0.600 mm,
	W =180.000 deg,	P =   0.000 deg,	R =    90.000 deg
};
P[4026]{
   GP1:
	UF : 1, UT : 1,		CONFIG : 'N U T, 0, 0, 1',
	X =  28.000  mm,	Y =  73.000  mm,	Z =   15.000 mm,
	W =180.000 deg,	P =   0.000 deg,	R =    90.000 deg
};
P[4027]{
   GP1:
	UF : 1, UT : 1,		CONFIG : 'N U T, 0, 0, 1',
	X =  31.000  mm,	Y =  73.000  mm,	Z =   15.000 mm,
	W =180.000 deg,	P =   0.000 deg,	R =    90.000 deg
};
P[4028]{
   GP1:
	UF : 1, UT : 1,		CONFIG : 'N U T, 0, 0, 1',
	X =  31.000  mm,	Y =  73.000  mm,	Z =   0.600 mm,
	W =180.000 deg,	P =   0.000 deg,	R =    90.000 deg
};
P[4029]{
   GP1:
	UF : 1, UT : 1,		CONFIG : 'N U T, 0, 0, 1',
	X =  31.000  mm,	Y =  73.000  mm,	Z =   15.000 mm,
	W =180.000 deg,	P =   0.000 deg,	R =    90.000 deg
};
P[4030]{
   GP1:
	UF : 1, UT : 1,		CONFIG : 'N U T, 0, 0, 1',
	X =  37.000  mm,	Y =  73.000  mm,	Z =   15.000 mm,
	W =180.000 deg,	P =   0.000 deg,	R =    90.000 deg
};
P[4031]{
   GP1:
	UF : 1, UT : 1,		CONFIG : 'N U T, 0, 0, 1',
	X =  37.000  mm,	Y =  73.000  mm,	Z =   0.600 mm,
	W =180.000 deg,	P =   0.000 deg,	R =    90.000 deg
};
P[4032]{
   GP1:
	UF : 1, UT : 1,		CONFIG : 'N U T, 0, 0, 1',
	X =  37.000  mm,	Y =  73.000  mm,	Z =   15.000 mm,
	W =180.000 deg,	P =   0.000 deg,	R =    90.000 deg
};
P[4033]{
   GP1:
	UF : 1, UT : 1,		CONFIG : 'N U T, 0, 0, 1',
	X =  40.000  mm,	Y =  73.000  mm,	Z =   15.000 mm,
	W =180.000 deg,	P =   0.000 deg,	R =    90.000 deg
};
P[4034]{
   GP1:
	UF : 1, UT : 1,		CONFIG : 'N U T, 0, 0, 1',
	X =  40.000  mm,	Y =  73.000  mm,	Z =   0.600 mm,
	W =180.000 deg,	P =   0.000 deg,	R =    90.000 deg
};
P[4035]{
   GP1:
	UF : 1, UT : 1,		CONFIG : 'N U T, 0, 0, 1',
	X =  40.000  mm,	Y =  73.000  mm,	Z =   15.000 mm,
	W =180.000 deg,	P =   0.000 deg,	R =    90.000 deg
};
P[4036]{
   GP1:
	UF : 1, UT : 1,		CONFIG : 'N U T, 0, 0, 1',
	X =  43.000  mm,	Y =  73.000  mm,	Z =   15.000 mm,
	W =180.000 deg,	P =   0.000 deg,	R =    90.000 deg
};
P[4037]{
   GP1:
	UF : 1, UT : 1,		CONFIG : 'N U T, 0, 0, 1',
	X =  43.000  mm,	Y =  73.000  mm,	Z =   0.600 mm,
	W =180.000 deg,	P =   0.000 deg,	R =    90.000 deg
};
P[4038]{
   GP1:
	UF : 1, UT : 1,		CONFIG : 'N U T, 0, 0, 1',
	X =  43.000  mm,	Y =  73.000  mm,	Z =   15.000 mm,
	W =180.000 deg,	P =   0.000 deg,	R =    90.000 deg
};
P[4039]{
   GP1:
	UF : 1, UT : 1,		CONFIG : 'N U T, 0, 0, 1',
	X =  46.000  mm,	Y =  73.000  mm,	Z =   15.000 mm,
	W =180.000 deg,	P =   0.000 deg,	R =    90.000 deg
};
P[4040]{
   GP1:
	UF : 1, UT : 1,		CONFIG : 'N U T, 0, 0, 1',
	X =  46.000  mm,	Y =  73.000  mm,	Z =   0.600 mm,
	W =180.000 deg,	P =   0.000 deg,	R =    90.000 deg
};
P[4041]{
   GP1:
	UF : 1, UT : 1,		CONFIG : 'N U T, 0, 0, 1',
	X =  46.000  mm,	Y =  73.000  mm,	Z =   15.000 mm,
	W =180.000 deg,	P =   0.000 deg,	R =    90.000 deg
};
P[4042]{
   GP1:
	UF : 1, UT : 1,		CONFIG : 'N U T, 0, 0, 1',
	X =  49.000  mm,	Y =  73.000  mm,	Z =   15.000 mm,
	W =180.000 deg,	P =   0.000 deg,	R =    90.000 deg
};
P[4043]{
   GP1:
	UF : 1, UT : 1,		CONFIG : 'N U T, 0, 0, 1',
	X =  49.000  mm,	Y =  73.000  mm,	Z =   0.600 mm,
	W =180.000 deg,	P =   0.000 deg,	R =    90.000 deg
};
P[4044]{
   GP1:
	UF : 1, UT : 1,		CONFIG : 'N U T, 0, 0, 1',
	X =  49.000  mm,	Y =  73.000  mm,	Z =   15.000 mm,
	W =180.000 deg,	P =   0.000 deg,	R =    90.000 deg
};
P[4045]{
   GP1:
	UF : 1, UT : 1,		CONFIG : 'N U T, 0, 0, 1',
	X =  52.000  mm,	Y =  73.000  mm,	Z =   15.000 mm,
	W =180.000 deg,	P =   0.000 deg,	R =    90.000 deg
};
P[4046]{
   GP1:
	UF : 1, UT : 1,		CONFIG : 'N U T, 0, 0, 1',
	X =  52.000  mm,	Y =  73.000  mm,	Z =   0.600 mm,
	W =180.000 deg,	P =   0.000 deg,	R =    90.000 deg
};
P[4047]{
   GP1:
	UF : 1, UT : 1,		CONFIG : 'N U T, 0, 0, 1',
	X =  52.000  mm,	Y =  73.000  mm,	Z =   15.000 mm,
	W =180.000 deg,	P =   0.000 deg,	R =    90.000 deg
};
P[4048]{
   GP1:
	UF : 1, UT : 1,		CONFIG : 'N U T, 0, 0, 1',
	X =  55.000  mm,	Y =  73.000  mm,	Z =   15.000 mm,
	W =180.000 deg,	P =   0.000 deg,	R =    90.000 deg
};
P[4049]{
   GP1:
	UF : 1, UT : 1,		CONFIG : 'N U T, 0, 0, 1',
	X =  55.000  mm,	Y =  73.000  mm,	Z =   0.600 mm,
	W =180.000 deg,	P =   0.000 deg,	R =    90.000 deg
};
P[4050]{
   GP1:
	UF : 1, UT : 1,		CONFIG : 'N U T, 0, 0, 1',
	X =  55.000  mm,	Y =  73.000  mm,	Z =   15.000 mm,
	W =180.000 deg,	P =   0.000 deg,	R =    90.000 deg
};
P[4051]{
   GP1:
	UF : 1, UT : 1,		CONFIG : 'N U T, 0, 0, 1',
	X =  58.000  mm,	Y =  73.000  mm,	Z =   15.000 mm,
	W =180.000 deg,	P =   0.000 deg,	R =    90.000 deg
};
P[4052]{
   GP1:
	UF : 1, UT : 1,		CONFIG : 'N U T, 0, 0, 1',
	X =  58.000  mm,	Y =  73.000  mm,	Z =   0.600 mm,
	W =180.000 deg,	P =   0.000 deg,	R =    90.000 deg
};
P[4053]{
   GP1:
	UF : 1, UT : 1,		CONFIG : 'N U T, 0, 0, 1',
	X =  58.000  mm,	Y =  73.000  mm,	Z =   15.000 mm,
	W =180.000 deg,	P =   0.000 deg,	R =    90.000 deg
};
P[4054]{
   GP1:
	UF : 1, UT : 1,		CONFIG : 'N U T, 0, 0, 1',
	X =  61.000  mm,	Y =  73.000  mm,	Z =   15.000 mm,
	W =180.000 deg,	P =   0.000 deg,	R =    90.000 deg
};
P[4055]{
   GP1:
	UF : 1, UT : 1,		CONFIG : 'N U T, 0, 0, 1',
	X =  61.000  mm,	Y =  73.000  mm,	Z =   0.600 mm,
	W =180.000 deg,	P =   0.000 deg,	R =    90.000 deg
};
P[4056]{
   GP1:
	UF : 1, UT : 1,		CONFIG : 'N U T, 0, 0, 1',
	X =  61.000  mm,	Y =  73.000  mm,	Z =   15.000 mm,
	W =180.000 deg,	P =   0.000 deg,	R =    90.000 deg
};
P[4057]{
   GP1:
	UF : 1, UT : 1,		CONFIG : 'N U T, 0, 0, 1',
	X =  64.000  mm,	Y =  73.000  mm,	Z =   15.000 mm,
	W =180.000 deg,	P =   0.000 deg,	R =    90.000 deg
};
P[4058]{
   GP1:
	UF : 1, UT : 1,		CONFIG : 'N U T, 0, 0, 1',
	X =  64.000  mm,	Y =  73.000  mm,	Z =   0.600 mm,
	W =180.000 deg,	P =   0.000 deg,	R =    90.000 deg
};
P[4059]{
   GP1:
	UF : 1, UT : 1,		CONFIG : 'N U T, 0, 0, 1',
	X =  64.000  mm,	Y =  73.000  mm,	Z =   15.000 mm,
	W =180.000 deg,	P =   0.000 deg,	R =    90.000 deg
};
P[4060]{
   GP1:
	UF : 1, UT : 1,		CONFIG : 'N U T, 0, 0, 1',
	X =  67.000  mm,	Y =  73.000  mm,	Z =   15.000 mm,
	W =180.000 deg,	P =   0.000 deg,	R =    90.000 deg
};
P[4061]{
   GP1:
	UF : 1, UT : 1,		CONFIG : 'N U T, 0, 0, 1',
	X =  67.000  mm,	Y =  73.000  mm,	Z =   0.600 mm,
	W =180.000 deg,	P =   0.000 deg,	R =    90.000 deg
};
P[4062]{
   GP1:
	UF : 1, UT : 1,		CONFIG : 'N U T, 0, 0, 1',
	X =  67.000  mm,	Y =  73.000  mm,	Z =   15.000 mm,
	W =180.000 deg,	P =   0.000 deg,	R =    90.000 deg
};
P[4063]{
   GP1:
	UF : 1, UT : 1,		CONFIG : 'N U T, 0, 0, 1',
	X =  70.000  mm,	Y =  73.000  mm,	Z =   15.000 mm,
	W =180.000 deg,	P =   0.000 deg,	R =    90.000 deg
};
P[4064]{
   GP1:
	UF : 1, UT : 1,		CONFIG : 'N U T, 0, 0, 1',
	X =  70.000  mm,	Y =  73.000  mm,	Z =   0.600 mm,
	W =180.000 deg,	P =   0.000 deg,	R =    90.000 deg
};
P[4065]{
   GP1:
	UF : 1, UT : 1,		CONFIG : 'N U T, 0, 0, 1',
	X =  70.000  mm,	Y =  73.000  mm,	Z =   15.000 mm,
	W =180.000 deg,	P =   0.000 deg,	R =    90.000 deg
};
P[4066]{
   GP1:
	UF : 1, UT : 1,		CONFIG : 'N U T, 0, 0, 1',
	X =  73.000  mm,	Y =  73.000  mm,	Z =   15.000 mm,
	W =180.000 deg,	P =   0.000 deg,	R =    90.000 deg
};
P[4067]{
   GP1:
	UF : 1, UT : 1,		CONFIG : 'N U T, 0, 0, 1',
	X =  73.000  mm,	Y =  73.000  mm,	Z =   0.600 mm,
	W =180.000 deg,	P =   0.000 deg,	R =    90.000 deg
};
P[4068]{
   GP1:
	UF : 1, UT : 1,		CONFIG : 'N U T, 0, 0, 1',
	X =  73.000  mm,	Y =  73.000  mm,	Z =   15.000 mm,
	W =180.000 deg,	P =   0.000 deg,	R =    90.000 deg
};
P[4072]{
   GP1:
	UF : 1, UT : 1,		CONFIG : 'N U T, 0, 0, 1',
	X =  82.000  mm,	Y =  73.000  mm,	Z =   15.000 mm,
	W =180.000 deg,	P =   0.000 deg,	R =    90.000 deg
};
P[4073]{
   GP1:
	UF : 1, UT : 1,		CONFIG : 'N U T, 0, 0, 1',
	X =  82.000  mm,	Y =  73.000  mm,	Z =   0.600 mm,
	W =180.000 deg,	P =   0.000 deg,	R =    90.000 deg
};
P[4074]{
   GP1:
	UF : 1, UT : 1,		CONFIG : 'N U T, 0, 0, 1',
	X =  82.000  mm,	Y =  73.000  mm,	Z =   15.000 mm,
	W =180.000 deg,	P =   0.000 deg,	R =    90.000 deg
};
P[4075]{
   GP1:
	UF : 1, UT : 1,		CONFIG : 'N U T, 0, 0, 1',
	X =  85.000  mm,	Y =  73.000  mm,	Z =   15.000 mm,
	W =180.000 deg,	P =   0.000 deg,	R =    90.000 deg
};
P[4076]{
   GP1:
	UF : 1, UT : 1,		CONFIG : 'N U T, 0, 0, 1',
	X =  85.000  mm,	Y =  73.000  mm,	Z =   0.600 mm,
	W =180.000 deg,	P =   0.000 deg,	R =    90.000 deg
};
P[4077]{
   GP1:
	UF : 1, UT : 1,		CONFIG : 'N U T, 0, 0, 1',
	X =  85.000  mm,	Y =  73.000  mm,	Z =   15.000 mm,
	W =180.000 deg,	P =   0.000 deg,	R =    90.000 deg
};
P[4078]{
   GP1:
	UF : 1, UT : 1,		CONFIG : 'N U T, 0, 0, 1',
	X =  88.000  mm,	Y =  73.000  mm,	Z =   15.000 mm,
	W =180.000 deg,	P =   0.000 deg,	R =    90.000 deg
};
P[4079]{
   GP1:
	UF : 1, UT : 1,		CONFIG : 'N U T, 0, 0, 1',
	X =  88.000  mm,	Y =  73.000  mm,	Z =   0.600 mm,
	W =180.000 deg,	P =   0.000 deg,	R =    90.000 deg
};
P[4080]{
   GP1:
	UF : 1, UT : 1,		CONFIG : 'N U T, 0, 0, 1',
	X =  88.000  mm,	Y =  73.000  mm,	Z =   15.000 mm,
	W =180.000 deg,	P =   0.000 deg,	R =    90.000 deg
};
P[4081]{
   GP1:
	UF : 1, UT : 1,		CONFIG : 'N U T, 0, 0, 1',
	X =  91.000  mm,	Y =  73.000  mm,	Z =   15.000 mm,
	W =180.000 deg,	P =   0.000 deg,	R =    90.000 deg
};
P[4082]{
   GP1:
	UF : 1, UT : 1,		CONFIG : 'N U T, 0, 0, 1',
	X =  91.000  mm,	Y =  73.000  mm,	Z =   0.600 mm,
	W =180.000 deg,	P =   0.000 deg,	R =    90.000 deg
};
P[4083]{
   GP1:
	UF : 1, UT : 1,		CONFIG : 'N U T, 0, 0, 1',
	X =  91.000  mm,	Y =  73.000  mm,	Z =   15.000 mm,
	W =180.000 deg,	P =   0.000 deg,	R =    90.000 deg
};
P[4084]{
   GP1:
	UF : 1, UT : 1,		CONFIG : 'N U T, 0, 0, 1',
	X =  94.000  mm,	Y =  73.000  mm,	Z =   15.000 mm,
	W =180.000 deg,	P =   0.000 deg,	R =    90.000 deg
};
P[4085]{
   GP1:
	UF : 1, UT : 1,		CONFIG : 'N U T, 0, 0, 1',
	X =  94.000  mm,	Y =  73.000  mm,	Z =   0.600 mm,
	W =180.000 deg,	P =   0.000 deg,	R =    90.000 deg
};
P[4086]{
   GP1:
	UF : 1, UT : 1,		CONFIG : 'N U T, 0, 0, 1',
	X =  94.000  mm,	Y =  73.000  mm,	Z =   15.000 mm,
	W =180.000 deg,	P =   0.000 deg,	R =    90.000 deg
};
P[4087]{
   GP1:
	UF : 1, UT : 1,		CONFIG : 'N U T, 0, 0, 1',
	X =  97.000  mm,	Y =  73.000  mm,	Z =   15.000 mm,
	W =180.000 deg,	P =   0.000 deg,	R =    90.000 deg
};
P[4088]{
   GP1:
	UF : 1, UT : 1,		CONFIG : 'N U T, 0, 0, 1',
	X =  97.000  mm,	Y =  73.000  mm,	Z =   0.600 mm,
	W =180.000 deg,	P =   0.000 deg,	R =    90.000 deg
};
P[4089]{
   GP1:
	UF : 1, UT : 1,		CONFIG : 'N U T, 0, 0, 1',
	X =  97.000  mm,	Y =  73.000  mm,	Z =   15.000 mm,
	W =180.000 deg,	P =   0.000 deg,	R =    90.000 deg
};
P[4090]{
   GP1:
	UF : 1, UT : 1,		CONFIG : 'N U T, 0, 0, 1',
	X =  100.000  mm,	Y =  73.000  mm,	Z =   15.000 mm,
	W =180.000 deg,	P =   0.000 deg,	R =    90.000 deg
};
P[4091]{
   GP1:
	UF : 1, UT : 1,		CONFIG : 'N U T, 0, 0, 1',
	X =  100.000  mm,	Y =  73.000  mm,	Z =   0.600 mm,
	W =180.000 deg,	P =   0.000 deg,	R =    90.000 deg
};
P[4092]{
   GP1:
	UF : 1, UT : 1,		CONFIG : 'N U T, 0, 0, 1',
	X =  100.000  mm,	Y =  73.000  mm,	Z =   15.000 mm,
	W =180.000 deg,	P =   0.000 deg,	R =    90.000 deg
};
P[4093]{
   GP1:
	UF : 1, UT : 1,		CONFIG : 'N U T, 0, 0, 1',
	X =  103.000  mm,	Y =  73.000  mm,	Z =   15.000 mm,
	W =180.000 deg,	P =   0.000 deg,	R =    90.000 deg
};
P[4094]{
   GP1:
	UF : 1, UT : 1,		CONFIG : 'N U T, 0, 0, 1',
	X =  103.000  mm,	Y =  73.000  mm,	Z =   0.600 mm,
	W =180.000 deg,	P =   0.000 deg,	R =    90.000 deg
};
P[4095]{
   GP1:
	UF : 1, UT : 1,		CONFIG : 'N U T, 0, 0, 1',
	X =  103.000  mm,	Y =  73.000  mm,	Z =   15.000 mm,
	W =180.000 deg,	P =   0.000 deg,	R =    90.000 deg
};
P[4096]{
   GP1:
	UF : 1, UT : 1,		CONFIG : 'N U T, 0, 0, 1',
	X =  106.000  mm,	Y =  73.000  mm,	Z =   15.000 mm,
	W =180.000 deg,	P =   0.000 deg,	R =    90.000 deg
};
P[4097]{
   GP1:
	UF : 1, UT : 1,		CONFIG : 'N U T, 0, 0, 1',
	X =  106.000  mm,	Y =  73.000  mm,	Z =   0.600 mm,
	W =180.000 deg,	P =   0.000 deg,	R =    90.000 deg
};
P[4098]{
   GP1:
	UF : 1, UT : 1,		CONFIG : 'N U T, 0, 0, 1',
	X =  106.000  mm,	Y =  73.000  mm,	Z =   15.000 mm,
	W =180.000 deg,	P =   0.000 deg,	R =    90.000 deg
};
P[4099]{
   GP1:
	UF : 1, UT : 1,		CONFIG : 'N U T, 0, 0, 1',
	X =  109.000  mm,	Y =  73.000  mm,	Z =   15.000 mm,
	W =180.000 deg,	P =   0.000 deg,	R =    90.000 deg
};
P[4100]{
   GP1:
	UF : 1, UT : 1,		CONFIG : 'N U T, 0, 0, 1',
	X =  109.000  mm,	Y =  73.000  mm,	Z =   0.600 mm,
	W =180.000 deg,	P =   0.000 deg,	R =    90.000 deg
};
P[4101]{
   GP1:
	UF : 1, UT : 1,		CONFIG : 'N U T, 0, 0, 1',
	X =  109.000  mm,	Y =  73.000  mm,	Z =   15.000 mm,
	W =180.000 deg,	P =   0.000 deg,	R =    90.000 deg
};
P[4102]{
   GP1:
	UF : 1, UT : 1,		CONFIG : 'N U T, 0, 0, 1',
	X =  112.000  mm,	Y =  73.000  mm,	Z =   15.000 mm,
	W =180.000 deg,	P =   0.000 deg,	R =    90.000 deg
};
P[4103]{
   GP1:
	UF : 1, UT : 1,		CONFIG : 'N U T, 0, 0, 1',
	X =  112.000  mm,	Y =  73.000  mm,	Z =   0.600 mm,
	W =180.000 deg,	P =   0.000 deg,	R =    90.000 deg
};
P[4104]{
   GP1:
	UF : 1, UT : 1,		CONFIG : 'N U T, 0, 0, 1',
	X =  112.000  mm,	Y =  73.000  mm,	Z =   15.000 mm,
	W =180.000 deg,	P =   0.000 deg,	R =    90.000 deg
};
P[4105]{
   GP1:
	UF : 1, UT : 1,		CONFIG : 'N U T, 0, 0, 1',
	X =  115.000  mm,	Y =  73.000  mm,	Z =   15.000 mm,
	W =180.000 deg,	P =   0.000 deg,	R =    90.000 deg
};
P[4106]{
   GP1:
	UF : 1, UT : 1,		CONFIG : 'N U T, 0, 0, 1',
	X =  115.000  mm,	Y =  73.000  mm,	Z =   0.600 mm,
	W =180.000 deg,	P =   0.000 deg,	R =    90.000 deg
};
P[4107]{
   GP1:
	UF : 1, UT : 1,		CONFIG : 'N U T, 0, 0, 1',
	X =  115.000  mm,	Y =  73.000  mm,	Z =   15.000 mm,
	W =180.000 deg,	P =   0.000 deg,	R =    90.000 deg
};
P[4108]{
   GP1:
	UF : 1, UT : 1,		CONFIG : 'N U T, 0, 0, 1',
	X =  133.000  mm,	Y =  73.000  mm,	Z =   15.000 mm,
	W =180.000 deg,	P =   0.000 deg,	R =    90.000 deg
};
P[4109]{
   GP1:
	UF : 1, UT : 1,		CONFIG : 'N U T, 0, 0, 1',
	X =  133.000  mm,	Y =  73.000  mm,	Z =   0.600 mm,
	W =180.000 deg,	P =   0.000 deg,	R =    90.000 deg
};
P[4110]{
   GP1:
	UF : 1, UT : 1,		CONFIG : 'N U T, 0, 0, 1',
	X =  133.000  mm,	Y =  73.000  mm,	Z =   15.000 mm,
	W =180.000 deg,	P =   0.000 deg,	R =    90.000 deg
};
P[4111]{
   GP1:
	UF : 1, UT : 1,		CONFIG : 'N U T, 0, 0, 1',
	X =  139.000  mm,	Y =  73.000  mm,	Z =   15.000 mm,
	W =180.000 deg,	P =   0.000 deg,	R =    90.000 deg
};
P[4112]{
   GP1:
	UF : 1, UT : 1,		CONFIG : 'N U T, 0, 0, 1',
	X =  139.000  mm,	Y =  73.000  mm,	Z =   0.600 mm,
	W =180.000 deg,	P =   0.000 deg,	R =    90.000 deg
};
P[4113]{
   GP1:
	UF : 1, UT : 1,		CONFIG : 'N U T, 0, 0, 1',
	X =  139.000  mm,	Y =  73.000  mm,	Z =   15.000 mm,
	W =180.000 deg,	P =   0.000 deg,	R =    90.000 deg
};
P[4117]{
   GP1:
	UF : 1, UT : 1,		CONFIG : 'N U T, 0, 0, 1',
	X =  145.000  mm,	Y =  73.000  mm,	Z =   15.000 mm,
	W =180.000 deg,	P =   0.000 deg,	R =    90.000 deg
};
P[4118]{
   GP1:
	UF : 1, UT : 1,		CONFIG : 'N U T, 0, 0, 1',
	X =  145.000  mm,	Y =  73.000  mm,	Z =   0.600 mm,
	W =180.000 deg,	P =   0.000 deg,	R =    90.000 deg
};
P[4119]{
   GP1:
	UF : 1, UT : 1,		CONFIG : 'N U T, 0, 0, 1',
	X =  145.000  mm,	Y =  73.000  mm,	Z =   15.000 mm,
	W =180.000 deg,	P =   0.000 deg,	R =    90.000 deg
};
P[4126]{
   GP1:
	UF : 1, UT : 1,		CONFIG : 'N U T, 0, 0, 1',
	X =  172.000  mm,	Y =  73.000  mm,	Z =   15.000 mm,
	W =180.000 deg,	P =   0.000 deg,	R =    90.000 deg
};
P[4127]{
   GP1:
	UF : 1, UT : 1,		CONFIG : 'N U T, 0, 0, 1',
	X =  172.000  mm,	Y =  73.000  mm,	Z =   0.600 mm,
	W =180.000 deg,	P =   0.000 deg,	R =    90.000 deg
};
P[4128]{
   GP1:
	UF : 1, UT : 1,		CONFIG : 'N U T, 0, 0, 1',
	X =  172.000  mm,	Y =  73.000  mm,	Z =   15.000 mm,
	W =180.000 deg,	P =   0.000 deg,	R =    90.000 deg
};
P[4129]{
   GP1:
	UF : 1, UT : 1,		CONFIG : 'N U T, 0, 0, 1',
	X =  175.000  mm,	Y =  73.000  mm,	Z =   15.000 mm,
	W =180.000 deg,	P =   0.000 deg,	R =    90.000 deg
};
P[4130]{
   GP1:
	UF : 1, UT : 1,		CONFIG : 'N U T, 0, 0, 1',
	X =  175.000  mm,	Y =  73.000  mm,	Z =   0.600 mm,
	W =180.000 deg,	P =   0.000 deg,	R =    90.000 deg
};
P[4131]{
   GP1:
	UF : 1, UT : 1,		CONFIG : 'N U T, 0, 0, 1',
	X =  175.000  mm,	Y =  73.000  mm,	Z =   15.000 mm,
	W =180.000 deg,	P =   0.000 deg,	R =    90.000 deg
};
P[4132]{
   GP1:
	UF : 1, UT : 1,		CONFIG : 'N U T, 0, 0, 1',
	X =  178.000  mm,	Y =  73.000  mm,	Z =   15.000 mm,
	W =180.000 deg,	P =   0.000 deg,	R =    90.000 deg
};
P[4133]{
   GP1:
	UF : 1, UT : 1,		CONFIG : 'N U T, 0, 0, 1',
	X =  178.000  mm,	Y =  73.000  mm,	Z =   0.600 mm,
	W =180.000 deg,	P =   0.000 deg,	R =    90.000 deg
};
P[4134]{
   GP1:
	UF : 1, UT : 1,		CONFIG : 'N U T, 0, 0, 1',
	X =  178.000  mm,	Y =  73.000  mm,	Z =   15.000 mm,
	W =180.000 deg,	P =   0.000 deg,	R =    90.000 deg
};
P[4135]{
   GP1:
	UF : 1, UT : 1,		CONFIG : 'N U T, 0, 0, 1',
	X =  1.000  mm,	Y =  76.000  mm,	Z =   15.000 mm,
	W =180.000 deg,	P =   0.000 deg,	R =    90.000 deg
};
P[4136]{
   GP1:
	UF : 1, UT : 1,		CONFIG : 'N U T, 0, 0, 1',
	X =  1.000  mm,	Y =  76.000  mm,	Z =   0.600 mm,
	W =180.000 deg,	P =   0.000 deg,	R =    90.000 deg
};
P[4137]{
   GP1:
	UF : 1, UT : 1,		CONFIG : 'N U T, 0, 0, 1',
	X =  1.000  mm,	Y =  76.000  mm,	Z =   15.000 mm,
	W =180.000 deg,	P =   0.000 deg,	R =    90.000 deg
};
P[4138]{
   GP1:
	UF : 1, UT : 1,		CONFIG : 'N U T, 0, 0, 1',
	X =  4.000  mm,	Y =  76.000  mm,	Z =   15.000 mm,
	W =180.000 deg,	P =   0.000 deg,	R =    90.000 deg
};
P[4139]{
   GP1:
	UF : 1, UT : 1,		CONFIG : 'N U T, 0, 0, 1',
	X =  4.000  mm,	Y =  76.000  mm,	Z =   0.600 mm,
	W =180.000 deg,	P =   0.000 deg,	R =    90.000 deg
};
P[4140]{
   GP1:
	UF : 1, UT : 1,		CONFIG : 'N U T, 0, 0, 1',
	X =  4.000  mm,	Y =  76.000  mm,	Z =   15.000 mm,
	W =180.000 deg,	P =   0.000 deg,	R =    90.000 deg
};
P[4141]{
   GP1:
	UF : 1, UT : 1,		CONFIG : 'N U T, 0, 0, 1',
	X =  7.000  mm,	Y =  76.000  mm,	Z =   15.000 mm,
	W =180.000 deg,	P =   0.000 deg,	R =    90.000 deg
};
P[4142]{
   GP1:
	UF : 1, UT : 1,		CONFIG : 'N U T, 0, 0, 1',
	X =  7.000  mm,	Y =  76.000  mm,	Z =   0.600 mm,
	W =180.000 deg,	P =   0.000 deg,	R =    90.000 deg
};
P[4143]{
   GP1:
	UF : 1, UT : 1,		CONFIG : 'N U T, 0, 0, 1',
	X =  7.000  mm,	Y =  76.000  mm,	Z =   15.000 mm,
	W =180.000 deg,	P =   0.000 deg,	R =    90.000 deg
};
P[4150]{
   GP1:
	UF : 1, UT : 1,		CONFIG : 'N U T, 0, 0, 1',
	X =  25.000  mm,	Y =  76.000  mm,	Z =   15.000 mm,
	W =180.000 deg,	P =   0.000 deg,	R =    90.000 deg
};
P[4151]{
   GP1:
	UF : 1, UT : 1,		CONFIG : 'N U T, 0, 0, 1',
	X =  25.000  mm,	Y =  76.000  mm,	Z =   0.600 mm,
	W =180.000 deg,	P =   0.000 deg,	R =    90.000 deg
};
P[4152]{
   GP1:
	UF : 1, UT : 1,		CONFIG : 'N U T, 0, 0, 1',
	X =  25.000  mm,	Y =  76.000  mm,	Z =   15.000 mm,
	W =180.000 deg,	P =   0.000 deg,	R =    90.000 deg
};
P[4153]{
   GP1:
	UF : 1, UT : 1,		CONFIG : 'N U T, 0, 0, 1',
	X =  28.000  mm,	Y =  76.000  mm,	Z =   15.000 mm,
	W =180.000 deg,	P =   0.000 deg,	R =    90.000 deg
};
P[4154]{
   GP1:
	UF : 1, UT : 1,		CONFIG : 'N U T, 0, 0, 1',
	X =  28.000  mm,	Y =  76.000  mm,	Z =   0.600 mm,
	W =180.000 deg,	P =   0.000 deg,	R =    90.000 deg
};
P[4155]{
   GP1:
	UF : 1, UT : 1,		CONFIG : 'N U T, 0, 0, 1',
	X =  28.000  mm,	Y =  76.000  mm,	Z =   15.000 mm,
	W =180.000 deg,	P =   0.000 deg,	R =    90.000 deg
};
P[4156]{
   GP1:
	UF : 1, UT : 1,		CONFIG : 'N U T, 0, 0, 1',
	X =  31.000  mm,	Y =  76.000  mm,	Z =   15.000 mm,
	W =180.000 deg,	P =   0.000 deg,	R =    90.000 deg
};
P[4157]{
   GP1:
	UF : 1, UT : 1,		CONFIG : 'N U T, 0, 0, 1',
	X =  31.000  mm,	Y =  76.000  mm,	Z =   0.600 mm,
	W =180.000 deg,	P =   0.000 deg,	R =    90.000 deg
};
P[4158]{
   GP1:
	UF : 1, UT : 1,		CONFIG : 'N U T, 0, 0, 1',
	X =  31.000  mm,	Y =  76.000  mm,	Z =   15.000 mm,
	W =180.000 deg,	P =   0.000 deg,	R =    90.000 deg
};
P[4159]{
   GP1:
	UF : 1, UT : 1,		CONFIG : 'N U T, 0, 0, 1',
	X =  34.000  mm,	Y =  76.000  mm,	Z =   15.000 mm,
	W =180.000 deg,	P =   0.000 deg,	R =    90.000 deg
};
P[4160]{
   GP1:
	UF : 1, UT : 1,		CONFIG : 'N U T, 0, 0, 1',
	X =  34.000  mm,	Y =  76.000  mm,	Z =   0.600 mm,
	W =180.000 deg,	P =   0.000 deg,	R =    90.000 deg
};
P[4161]{
   GP1:
	UF : 1, UT : 1,		CONFIG : 'N U T, 0, 0, 1',
	X =  34.000  mm,	Y =  76.000  mm,	Z =   15.000 mm,
	W =180.000 deg,	P =   0.000 deg,	R =    90.000 deg
};
P[4162]{
   GP1:
	UF : 1, UT : 1,		CONFIG : 'N U T, 0, 0, 1',
	X =  37.000  mm,	Y =  76.000  mm,	Z =   15.000 mm,
	W =180.000 deg,	P =   0.000 deg,	R =    90.000 deg
};
P[4163]{
   GP1:
	UF : 1, UT : 1,		CONFIG : 'N U T, 0, 0, 1',
	X =  37.000  mm,	Y =  76.000  mm,	Z =   0.600 mm,
	W =180.000 deg,	P =   0.000 deg,	R =    90.000 deg
};
P[4164]{
   GP1:
	UF : 1, UT : 1,		CONFIG : 'N U T, 0, 0, 1',
	X =  37.000  mm,	Y =  76.000  mm,	Z =   15.000 mm,
	W =180.000 deg,	P =   0.000 deg,	R =    90.000 deg
};
P[4165]{
   GP1:
	UF : 1, UT : 1,		CONFIG : 'N U T, 0, 0, 1',
	X =  40.000  mm,	Y =  76.000  mm,	Z =   15.000 mm,
	W =180.000 deg,	P =   0.000 deg,	R =    90.000 deg
};
P[4166]{
   GP1:
	UF : 1, UT : 1,		CONFIG : 'N U T, 0, 0, 1',
	X =  40.000  mm,	Y =  76.000  mm,	Z =   0.600 mm,
	W =180.000 deg,	P =   0.000 deg,	R =    90.000 deg
};
P[4167]{
   GP1:
	UF : 1, UT : 1,		CONFIG : 'N U T, 0, 0, 1',
	X =  40.000  mm,	Y =  76.000  mm,	Z =   15.000 mm,
	W =180.000 deg,	P =   0.000 deg,	R =    90.000 deg
};
P[4168]{
   GP1:
	UF : 1, UT : 1,		CONFIG : 'N U T, 0, 0, 1',
	X =  43.000  mm,	Y =  76.000  mm,	Z =   15.000 mm,
	W =180.000 deg,	P =   0.000 deg,	R =    90.000 deg
};
P[4169]{
   GP1:
	UF : 1, UT : 1,		CONFIG : 'N U T, 0, 0, 1',
	X =  43.000  mm,	Y =  76.000  mm,	Z =   0.600 mm,
	W =180.000 deg,	P =   0.000 deg,	R =    90.000 deg
};
P[4170]{
   GP1:
	UF : 1, UT : 1,		CONFIG : 'N U T, 0, 0, 1',
	X =  43.000  mm,	Y =  76.000  mm,	Z =   15.000 mm,
	W =180.000 deg,	P =   0.000 deg,	R =    90.000 deg
};
P[4171]{
   GP1:
	UF : 1, UT : 1,		CONFIG : 'N U T, 0, 0, 1',
	X =  46.000  mm,	Y =  76.000  mm,	Z =   15.000 mm,
	W =180.000 deg,	P =   0.000 deg,	R =    90.000 deg
};
P[4172]{
   GP1:
	UF : 1, UT : 1,		CONFIG : 'N U T, 0, 0, 1',
	X =  46.000  mm,	Y =  76.000  mm,	Z =   0.600 mm,
	W =180.000 deg,	P =   0.000 deg,	R =    90.000 deg
};
P[4173]{
   GP1:
	UF : 1, UT : 1,		CONFIG : 'N U T, 0, 0, 1',
	X =  46.000  mm,	Y =  76.000  mm,	Z =   15.000 mm,
	W =180.000 deg,	P =   0.000 deg,	R =    90.000 deg
};
P[4174]{
   GP1:
	UF : 1, UT : 1,		CONFIG : 'N U T, 0, 0, 1',
	X =  49.000  mm,	Y =  76.000  mm,	Z =   15.000 mm,
	W =180.000 deg,	P =   0.000 deg,	R =    90.000 deg
};
P[4175]{
   GP1:
	UF : 1, UT : 1,		CONFIG : 'N U T, 0, 0, 1',
	X =  49.000  mm,	Y =  76.000  mm,	Z =   0.600 mm,
	W =180.000 deg,	P =   0.000 deg,	R =    90.000 deg
};
P[4176]{
   GP1:
	UF : 1, UT : 1,		CONFIG : 'N U T, 0, 0, 1',
	X =  49.000  mm,	Y =  76.000  mm,	Z =   15.000 mm,
	W =180.000 deg,	P =   0.000 deg,	R =    90.000 deg
};
P[4177]{
   GP1:
	UF : 1, UT : 1,		CONFIG : 'N U T, 0, 0, 1',
	X =  52.000  mm,	Y =  76.000  mm,	Z =   15.000 mm,
	W =180.000 deg,	P =   0.000 deg,	R =    90.000 deg
};
P[4178]{
   GP1:
	UF : 1, UT : 1,		CONFIG : 'N U T, 0, 0, 1',
	X =  52.000  mm,	Y =  76.000  mm,	Z =   0.600 mm,
	W =180.000 deg,	P =   0.000 deg,	R =    90.000 deg
};
P[4179]{
   GP1:
	UF : 1, UT : 1,		CONFIG : 'N U T, 0, 0, 1',
	X =  52.000  mm,	Y =  76.000  mm,	Z =   15.000 mm,
	W =180.000 deg,	P =   0.000 deg,	R =    90.000 deg
};
P[4180]{
   GP1:
	UF : 1, UT : 1,		CONFIG : 'N U T, 0, 0, 1',
	X =  55.000  mm,	Y =  76.000  mm,	Z =   15.000 mm,
	W =180.000 deg,	P =   0.000 deg,	R =    90.000 deg
};
P[4181]{
   GP1:
	UF : 1, UT : 1,		CONFIG : 'N U T, 0, 0, 1',
	X =  55.000  mm,	Y =  76.000  mm,	Z =   0.600 mm,
	W =180.000 deg,	P =   0.000 deg,	R =    90.000 deg
};
P[4182]{
   GP1:
	UF : 1, UT : 1,		CONFIG : 'N U T, 0, 0, 1',
	X =  55.000  mm,	Y =  76.000  mm,	Z =   15.000 mm,
	W =180.000 deg,	P =   0.000 deg,	R =    90.000 deg
};
P[4183]{
   GP1:
	UF : 1, UT : 1,		CONFIG : 'N U T, 0, 0, 1',
	X =  58.000  mm,	Y =  76.000  mm,	Z =   15.000 mm,
	W =180.000 deg,	P =   0.000 deg,	R =    90.000 deg
};
P[4184]{
   GP1:
	UF : 1, UT : 1,		CONFIG : 'N U T, 0, 0, 1',
	X =  58.000  mm,	Y =  76.000  mm,	Z =   0.600 mm,
	W =180.000 deg,	P =   0.000 deg,	R =    90.000 deg
};
P[4185]{
   GP1:
	UF : 1, UT : 1,		CONFIG : 'N U T, 0, 0, 1',
	X =  58.000  mm,	Y =  76.000  mm,	Z =   15.000 mm,
	W =180.000 deg,	P =   0.000 deg,	R =    90.000 deg
};
P[4186]{
   GP1:
	UF : 1, UT : 1,		CONFIG : 'N U T, 0, 0, 1',
	X =  61.000  mm,	Y =  76.000  mm,	Z =   15.000 mm,
	W =180.000 deg,	P =   0.000 deg,	R =    90.000 deg
};
P[4187]{
   GP1:
	UF : 1, UT : 1,		CONFIG : 'N U T, 0, 0, 1',
	X =  61.000  mm,	Y =  76.000  mm,	Z =   0.600 mm,
	W =180.000 deg,	P =   0.000 deg,	R =    90.000 deg
};
P[4188]{
   GP1:
	UF : 1, UT : 1,		CONFIG : 'N U T, 0, 0, 1',
	X =  61.000  mm,	Y =  76.000  mm,	Z =   15.000 mm,
	W =180.000 deg,	P =   0.000 deg,	R =    90.000 deg
};
P[4189]{
   GP1:
	UF : 1, UT : 1,		CONFIG : 'N U T, 0, 0, 1',
	X =  64.000  mm,	Y =  76.000  mm,	Z =   15.000 mm,
	W =180.000 deg,	P =   0.000 deg,	R =    90.000 deg
};
P[4190]{
   GP1:
	UF : 1, UT : 1,		CONFIG : 'N U T, 0, 0, 1',
	X =  64.000  mm,	Y =  76.000  mm,	Z =   0.600 mm,
	W =180.000 deg,	P =   0.000 deg,	R =    90.000 deg
};
P[4191]{
   GP1:
	UF : 1, UT : 1,		CONFIG : 'N U T, 0, 0, 1',
	X =  64.000  mm,	Y =  76.000  mm,	Z =   15.000 mm,
	W =180.000 deg,	P =   0.000 deg,	R =    90.000 deg
};
P[4192]{
   GP1:
	UF : 1, UT : 1,		CONFIG : 'N U T, 0, 0, 1',
	X =  67.000  mm,	Y =  76.000  mm,	Z =   15.000 mm,
	W =180.000 deg,	P =   0.000 deg,	R =    90.000 deg
};
P[4193]{
   GP1:
	UF : 1, UT : 1,		CONFIG : 'N U T, 0, 0, 1',
	X =  67.000  mm,	Y =  76.000  mm,	Z =   0.600 mm,
	W =180.000 deg,	P =   0.000 deg,	R =    90.000 deg
};
P[4194]{
   GP1:
	UF : 1, UT : 1,		CONFIG : 'N U T, 0, 0, 1',
	X =  67.000  mm,	Y =  76.000  mm,	Z =   15.000 mm,
	W =180.000 deg,	P =   0.000 deg,	R =    90.000 deg
};
P[4195]{
   GP1:
	UF : 1, UT : 1,		CONFIG : 'N U T, 0, 0, 1',
	X =  70.000  mm,	Y =  76.000  mm,	Z =   15.000 mm,
	W =180.000 deg,	P =   0.000 deg,	R =    90.000 deg
};
P[4196]{
   GP1:
	UF : 1, UT : 1,		CONFIG : 'N U T, 0, 0, 1',
	X =  70.000  mm,	Y =  76.000  mm,	Z =   0.600 mm,
	W =180.000 deg,	P =   0.000 deg,	R =    90.000 deg
};
P[4197]{
   GP1:
	UF : 1, UT : 1,		CONFIG : 'N U T, 0, 0, 1',
	X =  70.000  mm,	Y =  76.000  mm,	Z =   15.000 mm,
	W =180.000 deg,	P =   0.000 deg,	R =    90.000 deg
};
P[4198]{
   GP1:
	UF : 1, UT : 1,		CONFIG : 'N U T, 0, 0, 1',
	X =  82.000  mm,	Y =  76.000  mm,	Z =   15.000 mm,
	W =180.000 deg,	P =   0.000 deg,	R =    90.000 deg
};
P[4199]{
   GP1:
	UF : 1, UT : 1,		CONFIG : 'N U T, 0, 0, 1',
	X =  82.000  mm,	Y =  76.000  mm,	Z =   0.600 mm,
	W =180.000 deg,	P =   0.000 deg,	R =    90.000 deg
};
P[4200]{
   GP1:
	UF : 1, UT : 1,		CONFIG : 'N U T, 0, 0, 1',
	X =  82.000  mm,	Y =  76.000  mm,	Z =   15.000 mm,
	W =180.000 deg,	P =   0.000 deg,	R =    90.000 deg
};
P[4201]{
   GP1:
	UF : 1, UT : 1,		CONFIG : 'N U T, 0, 0, 1',
	X =  85.000  mm,	Y =  76.000  mm,	Z =   15.000 mm,
	W =180.000 deg,	P =   0.000 deg,	R =    90.000 deg
};
P[4202]{
   GP1:
	UF : 1, UT : 1,		CONFIG : 'N U T, 0, 0, 1',
	X =  85.000  mm,	Y =  76.000  mm,	Z =   0.600 mm,
	W =180.000 deg,	P =   0.000 deg,	R =    90.000 deg
};
P[4203]{
   GP1:
	UF : 1, UT : 1,		CONFIG : 'N U T, 0, 0, 1',
	X =  85.000  mm,	Y =  76.000  mm,	Z =   15.000 mm,
	W =180.000 deg,	P =   0.000 deg,	R =    90.000 deg
};
P[4204]{
   GP1:
	UF : 1, UT : 1,		CONFIG : 'N U T, 0, 0, 1',
	X =  88.000  mm,	Y =  76.000  mm,	Z =   15.000 mm,
	W =180.000 deg,	P =   0.000 deg,	R =    90.000 deg
};
P[4205]{
   GP1:
	UF : 1, UT : 1,		CONFIG : 'N U T, 0, 0, 1',
	X =  88.000  mm,	Y =  76.000  mm,	Z =   0.600 mm,
	W =180.000 deg,	P =   0.000 deg,	R =    90.000 deg
};
P[4206]{
   GP1:
	UF : 1, UT : 1,		CONFIG : 'N U T, 0, 0, 1',
	X =  88.000  mm,	Y =  76.000  mm,	Z =   15.000 mm,
	W =180.000 deg,	P =   0.000 deg,	R =    90.000 deg
};
P[4207]{
   GP1:
	UF : 1, UT : 1,		CONFIG : 'N U T, 0, 0, 1',
	X =  91.000  mm,	Y =  76.000  mm,	Z =   15.000 mm,
	W =180.000 deg,	P =   0.000 deg,	R =    90.000 deg
};
P[4208]{
   GP1:
	UF : 1, UT : 1,		CONFIG : 'N U T, 0, 0, 1',
	X =  91.000  mm,	Y =  76.000  mm,	Z =   0.600 mm,
	W =180.000 deg,	P =   0.000 deg,	R =    90.000 deg
};
P[4209]{
   GP1:
	UF : 1, UT : 1,		CONFIG : 'N U T, 0, 0, 1',
	X =  91.000  mm,	Y =  76.000  mm,	Z =   15.000 mm,
	W =180.000 deg,	P =   0.000 deg,	R =    90.000 deg
};
P[4210]{
   GP1:
	UF : 1, UT : 1,		CONFIG : 'N U T, 0, 0, 1',
	X =  94.000  mm,	Y =  76.000  mm,	Z =   15.000 mm,
	W =180.000 deg,	P =   0.000 deg,	R =    90.000 deg
};
P[4211]{
   GP1:
	UF : 1, UT : 1,		CONFIG : 'N U T, 0, 0, 1',
	X =  94.000  mm,	Y =  76.000  mm,	Z =   0.600 mm,
	W =180.000 deg,	P =   0.000 deg,	R =    90.000 deg
};
P[4212]{
   GP1:
	UF : 1, UT : 1,		CONFIG : 'N U T, 0, 0, 1',
	X =  94.000  mm,	Y =  76.000  mm,	Z =   15.000 mm,
	W =180.000 deg,	P =   0.000 deg,	R =    90.000 deg
};
P[4213]{
   GP1:
	UF : 1, UT : 1,		CONFIG : 'N U T, 0, 0, 1',
	X =  97.000  mm,	Y =  76.000  mm,	Z =   15.000 mm,
	W =180.000 deg,	P =   0.000 deg,	R =    90.000 deg
};
P[4214]{
   GP1:
	UF : 1, UT : 1,		CONFIG : 'N U T, 0, 0, 1',
	X =  97.000  mm,	Y =  76.000  mm,	Z =   0.600 mm,
	W =180.000 deg,	P =   0.000 deg,	R =    90.000 deg
};
P[4215]{
   GP1:
	UF : 1, UT : 1,		CONFIG : 'N U T, 0, 0, 1',
	X =  97.000  mm,	Y =  76.000  mm,	Z =   15.000 mm,
	W =180.000 deg,	P =   0.000 deg,	R =    90.000 deg
};
P[4216]{
   GP1:
	UF : 1, UT : 1,		CONFIG : 'N U T, 0, 0, 1',
	X =  100.000  mm,	Y =  76.000  mm,	Z =   15.000 mm,
	W =180.000 deg,	P =   0.000 deg,	R =    90.000 deg
};
P[4217]{
   GP1:
	UF : 1, UT : 1,		CONFIG : 'N U T, 0, 0, 1',
	X =  100.000  mm,	Y =  76.000  mm,	Z =   0.600 mm,
	W =180.000 deg,	P =   0.000 deg,	R =    90.000 deg
};
P[4218]{
   GP1:
	UF : 1, UT : 1,		CONFIG : 'N U T, 0, 0, 1',
	X =  100.000  mm,	Y =  76.000  mm,	Z =   15.000 mm,
	W =180.000 deg,	P =   0.000 deg,	R =    90.000 deg
};
P[4219]{
   GP1:
	UF : 1, UT : 1,		CONFIG : 'N U T, 0, 0, 1',
	X =  103.000  mm,	Y =  76.000  mm,	Z =   15.000 mm,
	W =180.000 deg,	P =   0.000 deg,	R =    90.000 deg
};
P[4220]{
   GP1:
	UF : 1, UT : 1,		CONFIG : 'N U T, 0, 0, 1',
	X =  103.000  mm,	Y =  76.000  mm,	Z =   0.600 mm,
	W =180.000 deg,	P =   0.000 deg,	R =    90.000 deg
};
P[4221]{
   GP1:
	UF : 1, UT : 1,		CONFIG : 'N U T, 0, 0, 1',
	X =  103.000  mm,	Y =  76.000  mm,	Z =   15.000 mm,
	W =180.000 deg,	P =   0.000 deg,	R =    90.000 deg
};
P[4222]{
   GP1:
	UF : 1, UT : 1,		CONFIG : 'N U T, 0, 0, 1',
	X =  106.000  mm,	Y =  76.000  mm,	Z =   15.000 mm,
	W =180.000 deg,	P =   0.000 deg,	R =    90.000 deg
};
P[4223]{
   GP1:
	UF : 1, UT : 1,		CONFIG : 'N U T, 0, 0, 1',
	X =  106.000  mm,	Y =  76.000  mm,	Z =   0.600 mm,
	W =180.000 deg,	P =   0.000 deg,	R =    90.000 deg
};
P[4224]{
   GP1:
	UF : 1, UT : 1,		CONFIG : 'N U T, 0, 0, 1',
	X =  106.000  mm,	Y =  76.000  mm,	Z =   15.000 mm,
	W =180.000 deg,	P =   0.000 deg,	R =    90.000 deg
};
P[4225]{
   GP1:
	UF : 1, UT : 1,		CONFIG : 'N U T, 0, 0, 1',
	X =  109.000  mm,	Y =  76.000  mm,	Z =   15.000 mm,
	W =180.000 deg,	P =   0.000 deg,	R =    90.000 deg
};
P[4226]{
   GP1:
	UF : 1, UT : 1,		CONFIG : 'N U T, 0, 0, 1',
	X =  109.000  mm,	Y =  76.000  mm,	Z =   0.600 mm,
	W =180.000 deg,	P =   0.000 deg,	R =    90.000 deg
};
P[4227]{
   GP1:
	UF : 1, UT : 1,		CONFIG : 'N U T, 0, 0, 1',
	X =  109.000  mm,	Y =  76.000  mm,	Z =   15.000 mm,
	W =180.000 deg,	P =   0.000 deg,	R =    90.000 deg
};
P[4228]{
   GP1:
	UF : 1, UT : 1,		CONFIG : 'N U T, 0, 0, 1',
	X =  112.000  mm,	Y =  76.000  mm,	Z =   15.000 mm,
	W =180.000 deg,	P =   0.000 deg,	R =    90.000 deg
};
P[4229]{
   GP1:
	UF : 1, UT : 1,		CONFIG : 'N U T, 0, 0, 1',
	X =  112.000  mm,	Y =  76.000  mm,	Z =   0.600 mm,
	W =180.000 deg,	P =   0.000 deg,	R =    90.000 deg
};
P[4230]{
   GP1:
	UF : 1, UT : 1,		CONFIG : 'N U T, 0, 0, 1',
	X =  112.000  mm,	Y =  76.000  mm,	Z =   15.000 mm,
	W =180.000 deg,	P =   0.000 deg,	R =    90.000 deg
};
P[4231]{
   GP1:
	UF : 1, UT : 1,		CONFIG : 'N U T, 0, 0, 1',
	X =  115.000  mm,	Y =  76.000  mm,	Z =   15.000 mm,
	W =180.000 deg,	P =   0.000 deg,	R =    90.000 deg
};
P[4232]{
   GP1:
	UF : 1, UT : 1,		CONFIG : 'N U T, 0, 0, 1',
	X =  115.000  mm,	Y =  76.000  mm,	Z =   0.600 mm,
	W =180.000 deg,	P =   0.000 deg,	R =    90.000 deg
};
P[4233]{
   GP1:
	UF : 1, UT : 1,		CONFIG : 'N U T, 0, 0, 1',
	X =  115.000  mm,	Y =  76.000  mm,	Z =   15.000 mm,
	W =180.000 deg,	P =   0.000 deg,	R =    90.000 deg
};
P[4234]{
   GP1:
	UF : 1, UT : 1,		CONFIG : 'N U T, 0, 0, 1',
	X =  133.000  mm,	Y =  76.000  mm,	Z =   15.000 mm,
	W =180.000 deg,	P =   0.000 deg,	R =    90.000 deg
};
P[4235]{
   GP1:
	UF : 1, UT : 1,		CONFIG : 'N U T, 0, 0, 1',
	X =  133.000  mm,	Y =  76.000  mm,	Z =   0.600 mm,
	W =180.000 deg,	P =   0.000 deg,	R =    90.000 deg
};
P[4236]{
   GP1:
	UF : 1, UT : 1,		CONFIG : 'N U T, 0, 0, 1',
	X =  133.000  mm,	Y =  76.000  mm,	Z =   15.000 mm,
	W =180.000 deg,	P =   0.000 deg,	R =    90.000 deg
};
P[4237]{
   GP1:
	UF : 1, UT : 1,		CONFIG : 'N U T, 0, 0, 1',
	X =  136.000  mm,	Y =  76.000  mm,	Z =   15.000 mm,
	W =180.000 deg,	P =   0.000 deg,	R =    90.000 deg
};
P[4238]{
   GP1:
	UF : 1, UT : 1,		CONFIG : 'N U T, 0, 0, 1',
	X =  136.000  mm,	Y =  76.000  mm,	Z =   0.600 mm,
	W =180.000 deg,	P =   0.000 deg,	R =    90.000 deg
};
P[4239]{
   GP1:
	UF : 1, UT : 1,		CONFIG : 'N U T, 0, 0, 1',
	X =  136.000  mm,	Y =  76.000  mm,	Z =   15.000 mm,
	W =180.000 deg,	P =   0.000 deg,	R =    90.000 deg
};
P[4240]{
   GP1:
	UF : 1, UT : 1,		CONFIG : 'N U T, 0, 0, 1',
	X =  139.000  mm,	Y =  76.000  mm,	Z =   15.000 mm,
	W =180.000 deg,	P =   0.000 deg,	R =    90.000 deg
};
P[4241]{
   GP1:
	UF : 1, UT : 1,		CONFIG : 'N U T, 0, 0, 1',
	X =  139.000  mm,	Y =  76.000  mm,	Z =   0.600 mm,
	W =180.000 deg,	P =   0.000 deg,	R =    90.000 deg
};
P[4242]{
   GP1:
	UF : 1, UT : 1,		CONFIG : 'N U T, 0, 0, 1',
	X =  139.000  mm,	Y =  76.000  mm,	Z =   15.000 mm,
	W =180.000 deg,	P =   0.000 deg,	R =    90.000 deg
};
P[4243]{
   GP1:
	UF : 1, UT : 1,		CONFIG : 'N U T, 0, 0, 1',
	X =  142.000  mm,	Y =  76.000  mm,	Z =   15.000 mm,
	W =180.000 deg,	P =   0.000 deg,	R =    90.000 deg
};
P[4244]{
   GP1:
	UF : 1, UT : 1,		CONFIG : 'N U T, 0, 0, 1',
	X =  142.000  mm,	Y =  76.000  mm,	Z =   0.600 mm,
	W =180.000 deg,	P =   0.000 deg,	R =    90.000 deg
};
P[4245]{
   GP1:
	UF : 1, UT : 1,		CONFIG : 'N U T, 0, 0, 1',
	X =  142.000  mm,	Y =  76.000  mm,	Z =   15.000 mm,
	W =180.000 deg,	P =   0.000 deg,	R =    90.000 deg
};
P[4246]{
   GP1:
	UF : 1, UT : 1,		CONFIG : 'N U T, 0, 0, 1',
	X =  145.000  mm,	Y =  76.000  mm,	Z =   15.000 mm,
	W =180.000 deg,	P =   0.000 deg,	R =    90.000 deg
};
P[4247]{
   GP1:
	UF : 1, UT : 1,		CONFIG : 'N U T, 0, 0, 1',
	X =  145.000  mm,	Y =  76.000  mm,	Z =   0.600 mm,
	W =180.000 deg,	P =   0.000 deg,	R =    90.000 deg
};
P[4248]{
   GP1:
	UF : 1, UT : 1,		CONFIG : 'N U T, 0, 0, 1',
	X =  145.000  mm,	Y =  76.000  mm,	Z =   15.000 mm,
	W =180.000 deg,	P =   0.000 deg,	R =    90.000 deg
};
P[4249]{
   GP1:
	UF : 1, UT : 1,		CONFIG : 'N U T, 0, 0, 1',
	X =  169.000  mm,	Y =  76.000  mm,	Z =   15.000 mm,
	W =180.000 deg,	P =   0.000 deg,	R =    90.000 deg
};
P[4250]{
   GP1:
	UF : 1, UT : 1,		CONFIG : 'N U T, 0, 0, 1',
	X =  169.000  mm,	Y =  76.000  mm,	Z =   0.600 mm,
	W =180.000 deg,	P =   0.000 deg,	R =    90.000 deg
};
P[4251]{
   GP1:
	UF : 1, UT : 1,		CONFIG : 'N U T, 0, 0, 1',
	X =  169.000  mm,	Y =  76.000  mm,	Z =   15.000 mm,
	W =180.000 deg,	P =   0.000 deg,	R =    90.000 deg
};
P[4252]{
   GP1:
	UF : 1, UT : 1,		CONFIG : 'N U T, 0, 0, 1',
	X =  172.000  mm,	Y =  76.000  mm,	Z =   15.000 mm,
	W =180.000 deg,	P =   0.000 deg,	R =    90.000 deg
};
P[4253]{
   GP1:
	UF : 1, UT : 1,		CONFIG : 'N U T, 0, 0, 1',
	X =  172.000  mm,	Y =  76.000  mm,	Z =   0.600 mm,
	W =180.000 deg,	P =   0.000 deg,	R =    90.000 deg
};
P[4254]{
   GP1:
	UF : 1, UT : 1,		CONFIG : 'N U T, 0, 0, 1',
	X =  172.000  mm,	Y =  76.000  mm,	Z =   15.000 mm,
	W =180.000 deg,	P =   0.000 deg,	R =    90.000 deg
};
P[4255]{
   GP1:
	UF : 1, UT : 1,		CONFIG : 'N U T, 0, 0, 1',
	X =  175.000  mm,	Y =  76.000  mm,	Z =   15.000 mm,
	W =180.000 deg,	P =   0.000 deg,	R =    90.000 deg
};
P[4256]{
   GP1:
	UF : 1, UT : 1,		CONFIG : 'N U T, 0, 0, 1',
	X =  175.000  mm,	Y =  76.000  mm,	Z =   0.600 mm,
	W =180.000 deg,	P =   0.000 deg,	R =    90.000 deg
};
P[4257]{
   GP1:
	UF : 1, UT : 1,		CONFIG : 'N U T, 0, 0, 1',
	X =  175.000  mm,	Y =  76.000  mm,	Z =   15.000 mm,
	W =180.000 deg,	P =   0.000 deg,	R =    90.000 deg
};
P[4258]{
   GP1:
	UF : 1, UT : 1,		CONFIG : 'N U T, 0, 0, 1',
	X =  178.000  mm,	Y =  76.000  mm,	Z =   15.000 mm,
	W =180.000 deg,	P =   0.000 deg,	R =    90.000 deg
};
P[4259]{
   GP1:
	UF : 1, UT : 1,		CONFIG : 'N U T, 0, 0, 1',
	X =  178.000  mm,	Y =  76.000  mm,	Z =   0.600 mm,
	W =180.000 deg,	P =   0.000 deg,	R =    90.000 deg
};
P[4260]{
   GP1:
	UF : 1, UT : 1,		CONFIG : 'N U T, 0, 0, 1',
	X =  178.000  mm,	Y =  76.000  mm,	Z =   15.000 mm,
	W =180.000 deg,	P =   0.000 deg,	R =    90.000 deg
};
P[4261]{
   GP1:
	UF : 1, UT : 1,		CONFIG : 'N U T, 0, 0, 1',
	X =  1.000  mm,	Y =  79.000  mm,	Z =   15.000 mm,
	W =180.000 deg,	P =   0.000 deg,	R =    90.000 deg
};
P[4262]{
   GP1:
	UF : 1, UT : 1,		CONFIG : 'N U T, 0, 0, 1',
	X =  1.000  mm,	Y =  79.000  mm,	Z =   0.600 mm,
	W =180.000 deg,	P =   0.000 deg,	R =    90.000 deg
};
P[4263]{
   GP1:
	UF : 1, UT : 1,		CONFIG : 'N U T, 0, 0, 1',
	X =  1.000  mm,	Y =  79.000  mm,	Z =   15.000 mm,
	W =180.000 deg,	P =   0.000 deg,	R =    90.000 deg
};
P[4264]{
   GP1:
	UF : 1, UT : 1,		CONFIG : 'N U T, 0, 0, 1',
	X =  4.000  mm,	Y =  79.000  mm,	Z =   15.000 mm,
	W =180.000 deg,	P =   0.000 deg,	R =    90.000 deg
};
P[4265]{
   GP1:
	UF : 1, UT : 1,		CONFIG : 'N U T, 0, 0, 1',
	X =  4.000  mm,	Y =  79.000  mm,	Z =   0.600 mm,
	W =180.000 deg,	P =   0.000 deg,	R =    90.000 deg
};
P[4266]{
   GP1:
	UF : 1, UT : 1,		CONFIG : 'N U T, 0, 0, 1',
	X =  4.000  mm,	Y =  79.000  mm,	Z =   15.000 mm,
	W =180.000 deg,	P =   0.000 deg,	R =    90.000 deg
};
P[4294]{
   GP1:
	UF : 1, UT : 1,		CONFIG : 'N U T, 0, 0, 1',
	X =  37.000  mm,	Y =  79.000  mm,	Z =   15.000 mm,
	W =180.000 deg,	P =   0.000 deg,	R =    90.000 deg
};
P[4295]{
   GP1:
	UF : 1, UT : 1,		CONFIG : 'N U T, 0, 0, 1',
	X =  37.000  mm,	Y =  79.000  mm,	Z =   0.600 mm,
	W =180.000 deg,	P =   0.000 deg,	R =    90.000 deg
};
P[4296]{
   GP1:
	UF : 1, UT : 1,		CONFIG : 'N U T, 0, 0, 1',
	X =  37.000  mm,	Y =  79.000  mm,	Z =   15.000 mm,
	W =180.000 deg,	P =   0.000 deg,	R =    90.000 deg
};
P[4297]{
   GP1:
	UF : 1, UT : 1,		CONFIG : 'N U T, 0, 0, 1',
	X =  40.000  mm,	Y =  79.000  mm,	Z =   15.000 mm,
	W =180.000 deg,	P =   0.000 deg,	R =    90.000 deg
};
P[4298]{
   GP1:
	UF : 1, UT : 1,		CONFIG : 'N U T, 0, 0, 1',
	X =  40.000  mm,	Y =  79.000  mm,	Z =   0.600 mm,
	W =180.000 deg,	P =   0.000 deg,	R =    90.000 deg
};
P[4299]{
   GP1:
	UF : 1, UT : 1,		CONFIG : 'N U T, 0, 0, 1',
	X =  40.000  mm,	Y =  79.000  mm,	Z =   15.000 mm,
	W =180.000 deg,	P =   0.000 deg,	R =    90.000 deg
};
P[4300]{
   GP1:
	UF : 1, UT : 1,		CONFIG : 'N U T, 0, 0, 1',
	X =  43.000  mm,	Y =  79.000  mm,	Z =   15.000 mm,
	W =180.000 deg,	P =   0.000 deg,	R =    90.000 deg
};
P[4301]{
   GP1:
	UF : 1, UT : 1,		CONFIG : 'N U T, 0, 0, 1',
	X =  43.000  mm,	Y =  79.000  mm,	Z =   0.600 mm,
	W =180.000 deg,	P =   0.000 deg,	R =    90.000 deg
};
P[4302]{
   GP1:
	UF : 1, UT : 1,		CONFIG : 'N U T, 0, 0, 1',
	X =  43.000  mm,	Y =  79.000  mm,	Z =   15.000 mm,
	W =180.000 deg,	P =   0.000 deg,	R =    90.000 deg
};
P[4303]{
   GP1:
	UF : 1, UT : 1,		CONFIG : 'N U T, 0, 0, 1',
	X =  46.000  mm,	Y =  79.000  mm,	Z =   15.000 mm,
	W =180.000 deg,	P =   0.000 deg,	R =    90.000 deg
};
P[4304]{
   GP1:
	UF : 1, UT : 1,		CONFIG : 'N U T, 0, 0, 1',
	X =  46.000  mm,	Y =  79.000  mm,	Z =   0.600 mm,
	W =180.000 deg,	P =   0.000 deg,	R =    90.000 deg
};
P[4305]{
   GP1:
	UF : 1, UT : 1,		CONFIG : 'N U T, 0, 0, 1',
	X =  46.000  mm,	Y =  79.000  mm,	Z =   15.000 mm,
	W =180.000 deg,	P =   0.000 deg,	R =    90.000 deg
};
P[4306]{
